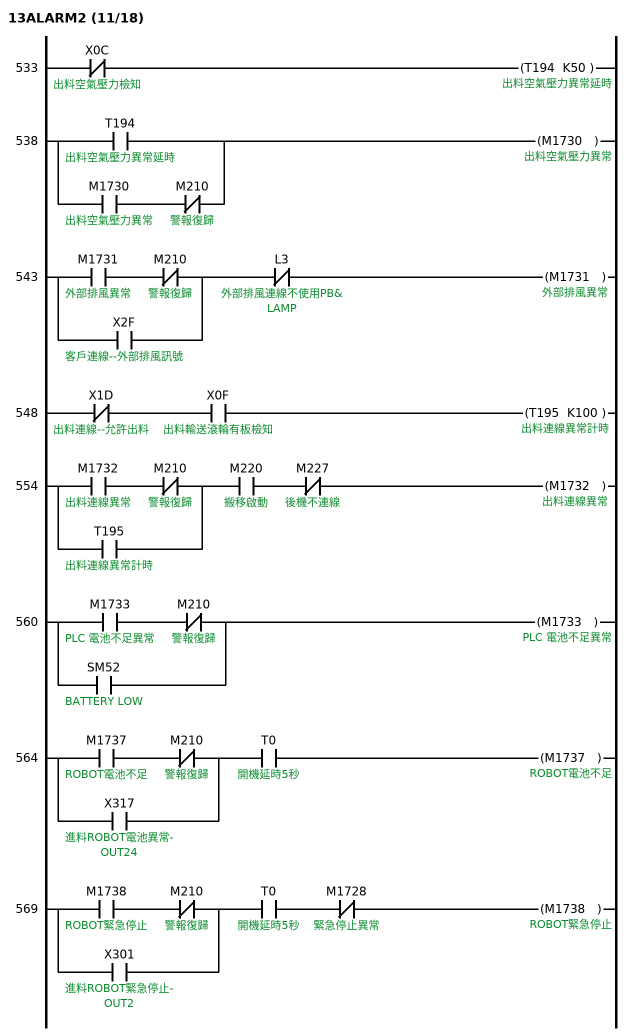
[picture p72: ladder of 13ALARM2, rungs at steps 533 to 569]
533   LDI     X0C  ; 出料空氣壓力檢知
      OUT     T194 K50  ; 出料空氣壓力異常延時
538   LD      T194  ; 出料空氣壓力異常延時
      LD      M1730  ; 出料空氣壓力異常
      ANI     M210  ; 警報復歸
      ORB
      OUT     M1730  ; 出料空氣壓力異常
543   LD      M1731  ; 外部排風異常
      ANI     M210  ; 警報復歸
      OR      X2F  ; 客戶連線--外部排風訊號
      ANI     L3  ; 外部排風連線不使用PB&LAMP
      OUT     M1731  ; 外部排風異常
548   LDI     X1D  ; 出料連線--允許出料
      AND     X0F  ; 出料輸送滾輪有板檢知
      OUT     T195 K100  ; 出料連線異常計時
554   LD      M1732  ; 出料連線異常
      ANI     M210  ; 警報復歸
      OR      T195  ; 出料連線異常計時
      AND     M220  ; 搬移啟動
      ANI     M227  ; 後機不連線
      OUT     M1732  ; 出料連線異常
560   LD      M1733  ; PLC 電池不足異常
      ANI     M210  ; 警報復歸
      OR      SM52  ; BATTERY LOW
      OUT     M1733  ; PLC 電池不足異常
564   LD      M1737  ; ROBOT電池不足
      ANI     M210  ; 警報復歸
      OR      X317  ; 進料ROBOT電池異常-OUT24
      AND     T0  ; 開機延時5秒
      OUT     M1737  ; ROBOT電池不足
569   LD      M1738  ; ROBOT緊急停止
      ANI     M210  ; 警報復歸
      OR      X301  ; 進料ROBOT緊急停止-OUT2
      AND     T0  ; 開機延時5秒
      ANI     M1728  ; 緊急停止異常
      OUT     M1738  ; ROBOT緊急停止
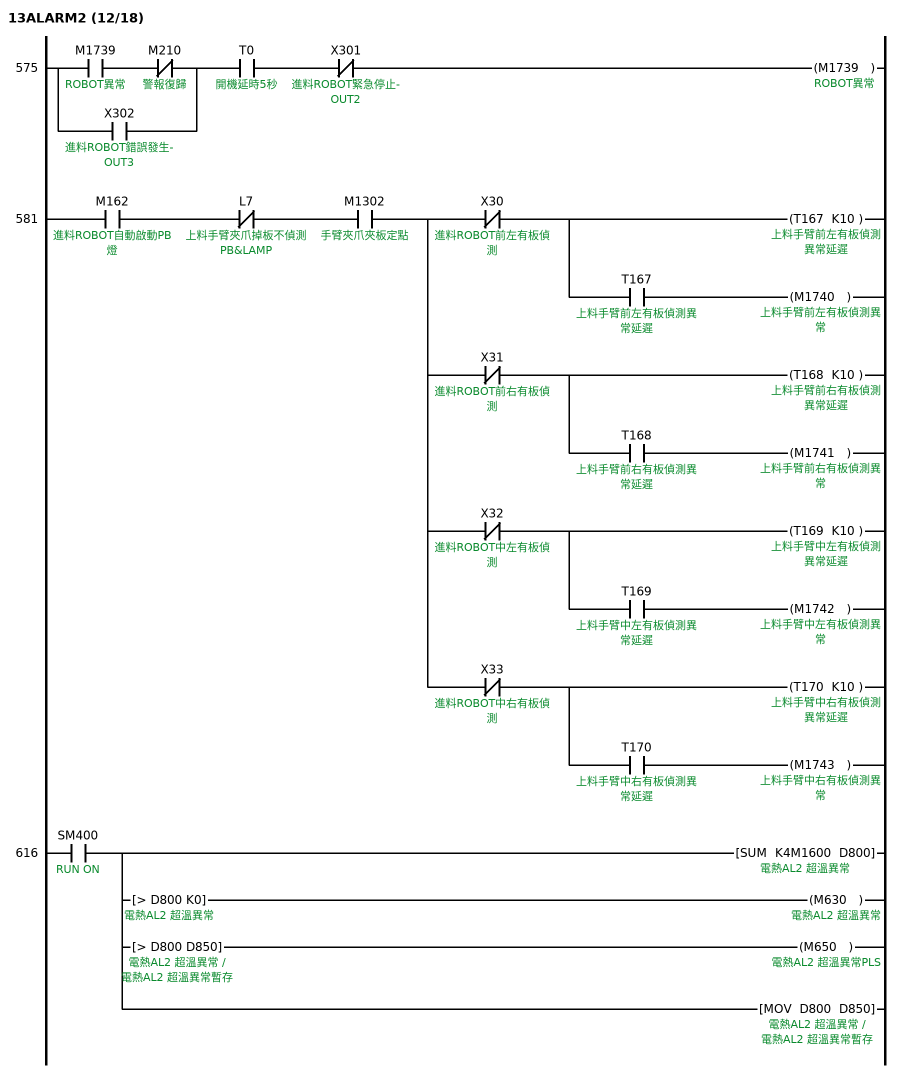
575   LD      M1739  ; ROBOT異常
      ANI     M210  ; 警報復歸
      OR      X302  ; 進料ROBOT錯誤發生-OUT3
      AND     T0  ; 開機延時5秒
      ANI     X301  ; 進料ROBOT緊急停止-OUT2
      OUT     M1739  ; ROBOT異常
581   LD      M162  ; 進料ROBOT自動啟動PB燈
      ANI     L7  ; 上料手臂夾爪掉板不偵測PB&LAMP
      AND     M1302  ; 手臂夾爪夾板定點
      MPS
      ANI     X30  ; 進料ROBOT前左有板偵測
      OUT     T167 K10  ; 上料手臂前左有板偵測異常延遲
      AND     T167  ; 上料手臂前左有板偵測異常延遲
      OUT     M1740  ; 上料手臂前左有板偵測異常
      MRD
      ANI     X31  ; 進料ROBOT前右有板偵測
      OUT     T168 K10  ; 上料手臂前右有板偵測異常延遲
      AND     T168  ; 上料手臂前右有板偵測異常延遲
      OUT     M1741  ; 上料手臂前右有板偵測異常
      MRD
      ANI     X32  ; 進料ROBOT中左有板偵測
      OUT     T169 K10  ; 上料手臂中左有板偵測異常延遲
      AND     T169  ; 上料手臂中左有板偵測異常延遲
      OUT     M1742  ; 上料手臂中左有板偵測異常
      MPP
      ANI     X33  ; 進料ROBOT中右有板偵測
      OUT     T170 K10  ; 上料手臂中右有板偵測異常延遲
      AND     T170  ; 上料手臂中右有板偵測異常延遲
      OUT     M1743  ; 上料手臂中右有板偵測異常
616   LD      SM400  ; RUN ON
      SUM     K4M1600 D800  ; #01 電熱AL2 超溫 / 電熱AL2 超溫異常
      MPS
      AND>    D800 K0  ; 電熱AL2 超溫異常
      OUT     M630  ; 電熱AL2 超溫異常
      MRD
      AND>    D800 D850  ; 電熱AL2 超溫異常 / 電熱AL2 超溫異常暫存
      OUT     M650  ; 電熱AL2 超溫異常PLS
      MPP
      MOV     D800 D850
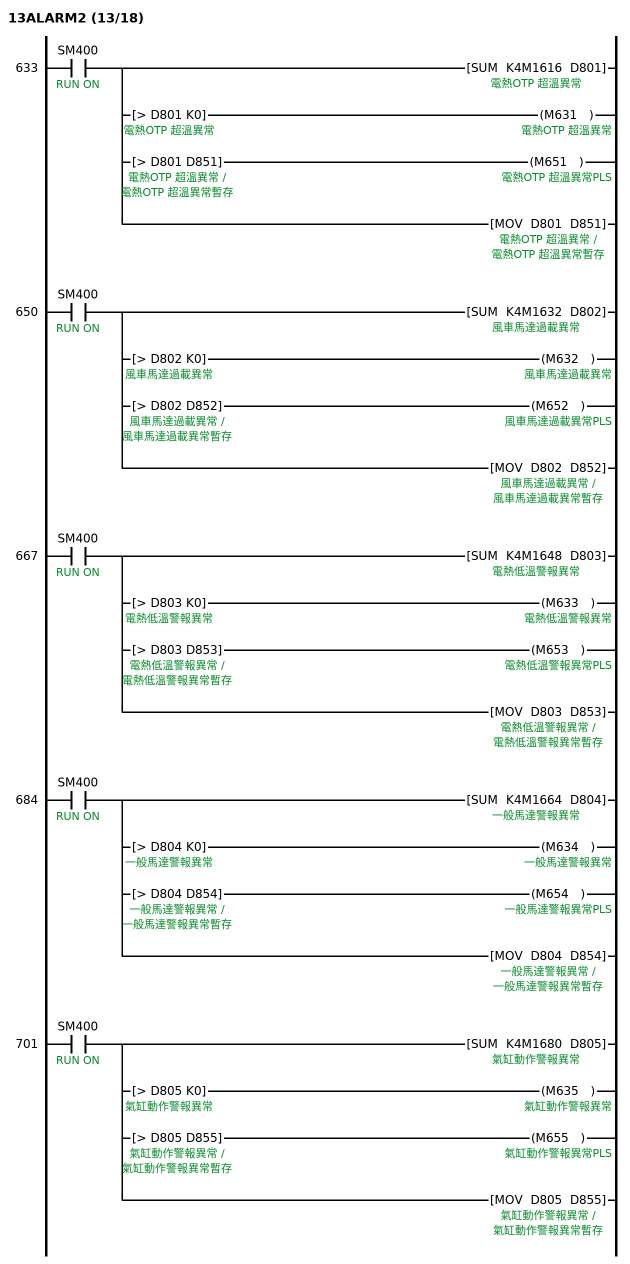
633   LD      SM400  ; RUN ON
      SUM     K4M1616 D801  ; #01 電熱OTP 超溫 / 電熱OTP 超溫異常
      MPS
      AND>    D801 K0  ; 電熱OTP 超溫異常
      OUT     M631  ; 電熱OTP 超溫異常
      MRD
      AND>    D801 D851  ; 電熱OTP 超溫異常 / 電熱OTP 超溫異常暫存
      OUT     M651  ; 電熱OTP 超溫異常PLS
      MPP
      MOV     D801 D851
650   LD      SM400  ; RUN ON
      SUM     K4M1632 D802  ; #01 風車過載 / 風車馬達過載異常
      MPS
      AND>    D802 K0  ; 風車馬達過載異常
      OUT     M632  ; 風車馬達過載異常
      MRD
      AND>    D802 D852  ; 風車馬達過載異常 / 風車馬達過載異常暫存
      OUT     M652  ; 風車馬達過載異常PLS
      MPP
      MOV     D802 D852
667   LD      SM400  ; RUN ON
      SUM     K4M1648 D803  ; #01 低溫警報 / 電熱低溫警報異常
      MPS
      AND>    D803 K0  ; 電熱低溫警報異常
      OUT     M633  ; 電熱低溫警報異常
      MRD
      AND>    D803 D853  ; 電熱低溫警報異常 / 電熱低溫警報異常暫存
      OUT     M653  ; 電熱低溫警報異常PLS
      MPP
      MOV     D803 D853
684   LD      SM400  ; RUN ON
      SUM     K4M1664 D804  ; 一般馬達警報異常
      MPS
      AND>    D804 K0  ; 一般馬達警報異常
      OUT     M634  ; 一般馬達警報異常
      MRD
      AND>    D804 D854  ; 一般馬達警報異常 / 一般馬達警報異常暫存
      OUT     M654  ; 一般馬達警報異常PLS
      MPP
      MOV     D804 D854
701   LD      SM400  ; RUN ON
      SUM     K4M1680 D805  ; 氣缸動作警報異常
      MPS
      AND>    D805 K0  ; 氣缸動作警報異常
      OUT     M635  ; 氣缸動作警報異常
      MRD
      AND>    D805 D855  ; 氣缸動作警報異常 / 氣缸動作警報異常暫存
      OUT     M655  ; 氣缸動作警報異常PLS
      MPP
      MOV     D805 D855
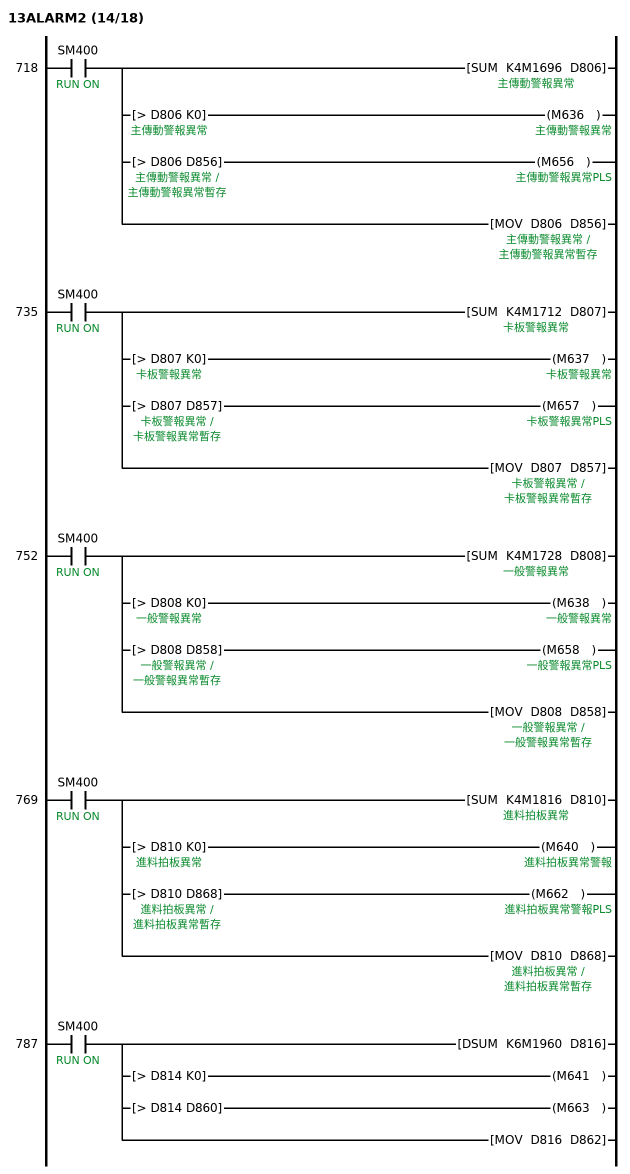
718   LD      SM400  ; RUN ON
      SUM     K4M1696 D806  ; 主傳動警報異常
      MPS
      AND>    D806 K0  ; 主傳動警報異常
      OUT     M636  ; 主傳動警報異常
      MRD
      AND>    D806 D856  ; 主傳動警報異常 / 主傳動警報異常暫存
      OUT     M656  ; 主傳動警報異常PLS
      MPP
      MOV     D806 D856
735   LD      SM400  ; RUN ON
      SUM     K4M1712 D807  ; 卡板警報異常
      MPS
      AND>    D807 K0  ; 卡板警報異常
      OUT     M637  ; 卡板警報異常
      MRD
      AND>    D807 D857  ; 卡板警報異常 / 卡板警報異常暫存
      OUT     M657  ; 卡板警報異常PLS
      MPP
      MOV     D807 D857
752   LD      SM400  ; RUN ON
      SUM     K4M1728 D808  ; 一般警報異常
      MPS
      AND>    D808 K0  ; 一般警報異常
      OUT     M638  ; 一般警報異常
      MRD
      AND>    D808 D858  ; 一般警報異常 / 一般警報異常暫存
      OUT     M658  ; 一般警報異常PLS
      MPP
      MOV     D808 D858
769   LD      SM400  ; RUN ON
      SUM     K4M1816 D810  ; 輸送機輸送變頻器異常-ALM / 進料拍板異常
      MPS
      AND>    D810 K0  ; 進料拍板異常
      OUT     M640  ; 進料拍板異常警報
      MRD
      AND>    D810 D868  ; 進料拍板異常 / 進料拍板異常暫存
      OUT     M662  ; 進料拍板異常警報PLS
      MPP
      MOV     D810 D868
787   LD      SM400  ; RUN ON
      DSUM    K6M1960 D816
      MPS
      AND>    D814 K0
      OUT     M641
      MRD
      AND>    D814 D860
      OUT     M663
      MPP
      MOV     D816 D862
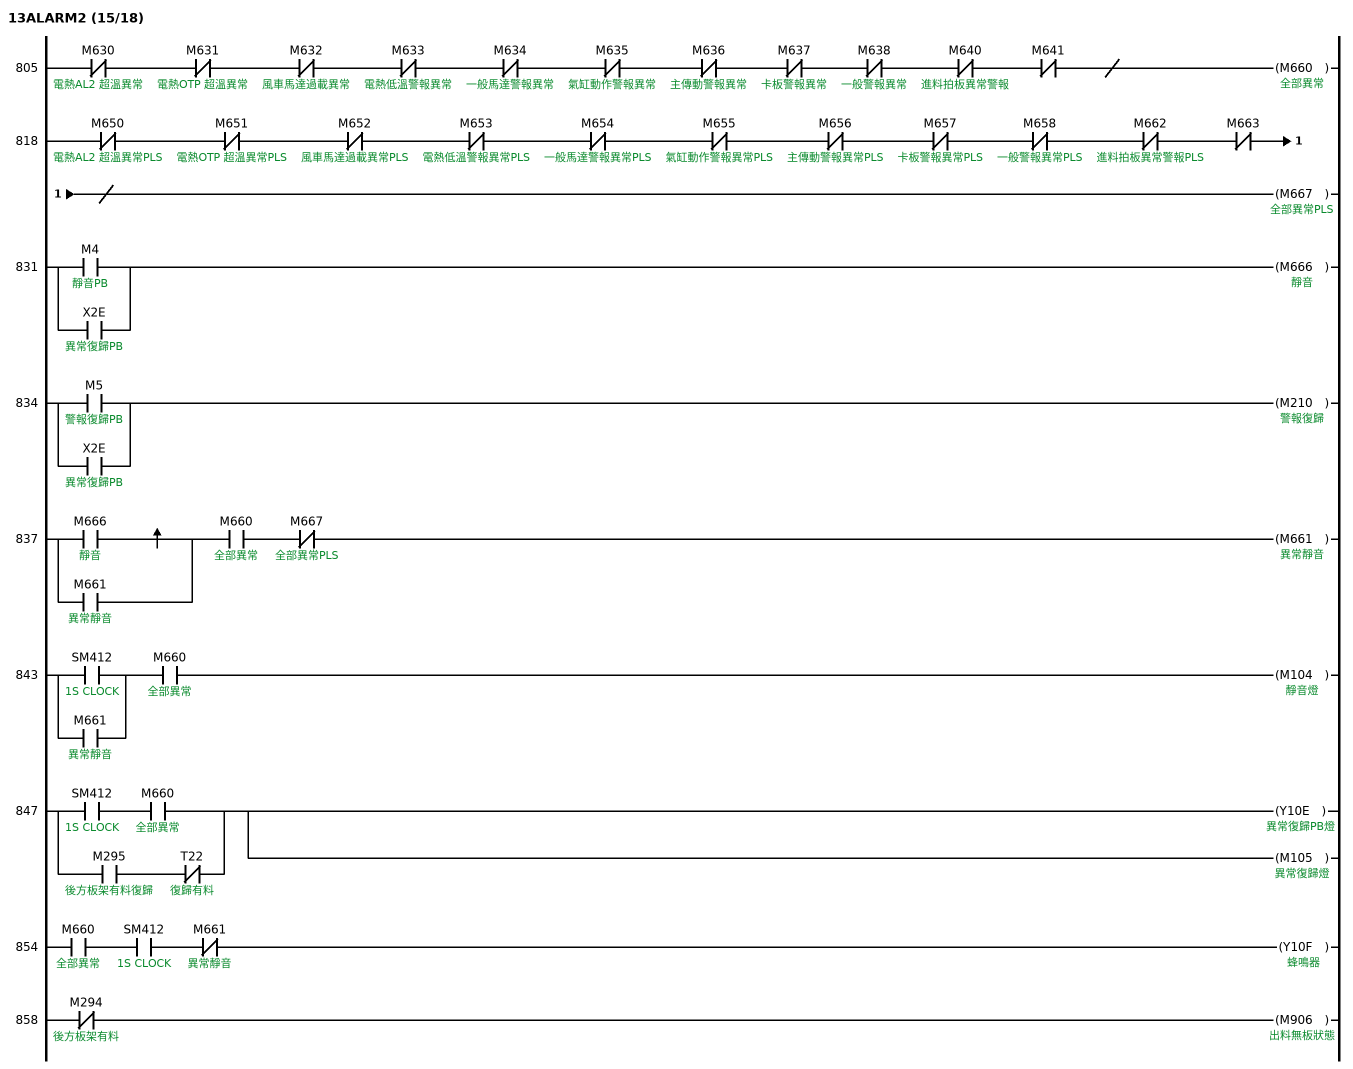
805   LDI     M630  ; 電熱AL2 超溫異常
      ANI     M631  ; 電熱OTP 超溫異常
      ANI     M632  ; 風車馬達過載異常
      ANI     M633  ; 電熱低溫警報異常
      ANI     M634  ; 一般馬達警報異常
      ANI     M635  ; 氣缸動作警報異常
      ANI     M636  ; 主傳動警報異常
      ANI     M637  ; 卡板警報異常
      ANI     M638  ; 一般警報異常
      ANI     M640  ; 進料拍板異常警報
      ANI     M641
      INV
      OUT     M660  ; 全部異常
818   LDI     M650  ; 電熱AL2 超溫異常PLS
      ANI     M651  ; 電熱OTP 超溫異常PLS
      ANI     M652  ; 風車馬達過載異常PLS
      ANI     M653  ; 電熱低溫警報異常PLS
      ANI     M654  ; 一般馬達警報異常PLS
      ANI     M655  ; 氣缸動作警報異常PLS
      ANI     M656  ; 主傳動警報異常PLS
      ANI     M657  ; 卡板警報異常PLS
      ANI     M658  ; 一般警報異常PLS
      ANI     M662  ; 進料拍板異常警報PLS
      ANI     M663
      INV
      OUT     M667  ; 全部異常PLS
831   LD      M4  ; 靜音PB
      OR      X2E  ; 異常復歸PB
      OUT     M666  ; 靜音
834   LD      M5  ; 警報復歸PB
      OR      X2E  ; 異常復歸PB
      OUT     M210  ; 警報復歸
837   LD      M666  ; 靜音
      MEP
      OR      M661  ; 異常靜音
      AND     M660  ; 全部異常
      ANI     M667  ; 全部異常PLS
      OUT     M661  ; 異常靜音
843   LD      SM412  ; 1S CLOCK
      OR      M661  ; 異常靜音
      AND     M660  ; 全部異常
      OUT     M104  ; 靜音燈
847   LD      SM412  ; 1S CLOCK
      AND     M660  ; 全部異常
      LD      M295  ; 後方板架有料復歸
      ANI     T22  ; 復歸有料
      ORB
      OUT     Y10E  ; 異常復歸PB燈
      OUT     M105  ; 異常復歸燈
854   LD      M660  ; 全部異常
      AND     SM412  ; 1S CLOCK
      ANI     M661  ; 異常靜音
      OUT     Y10F  ; 蜂鳴器
858   LDI     M294  ; 後方板架有料
      OUT     M906  ; 出料無板狀態
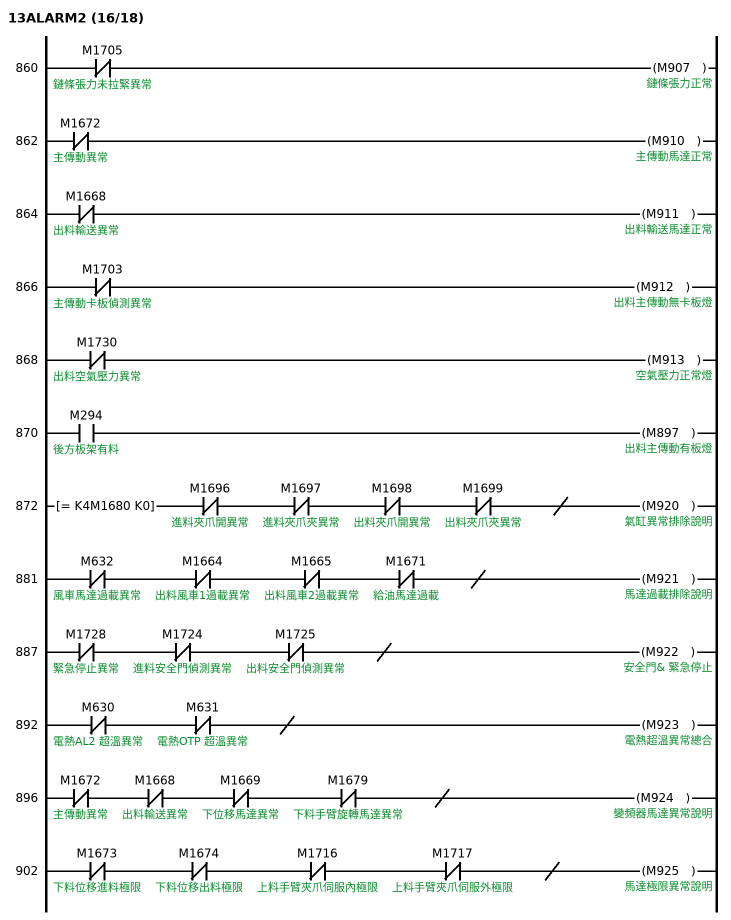
860   LDI     M1705  ; 鏈條張力未拉緊異常
      OUT     M907  ; 鏈條張力正常
862   LDI     M1672  ; 主傳動異常
      OUT     M910  ; 主傳動馬達正常
864   LDI     M1668  ; 出料輸送異常
      OUT     M911  ; 出料輸送馬達正常
866   LDI     M1703  ; 主傳動卡板偵測異常
      OUT     M912  ; 出料主傳動無卡板燈
868   LDI     M1730  ; 出料空氣壓力異常
      OUT     M913  ; 空氣壓力正常燈
870   LD      M294  ; 後方板架有料
      OUT     M897  ; 出料主傳動有板燈
872   LD=     K4M1680 K0  ; 上料手臂前夾爪放異常
      ANI     M1696  ; 進料夾爪開異常
      ANI     M1697  ; 進料夾爪夾異常
      ANI     M1698  ; 出料夾爪開異常
      ANI     M1699  ; 出料夾爪夾異常
      INV
      OUT     M920  ; 氣缸異常排除說明
881   LDI     M632  ; 風車馬達過載異常
      ANI     M1664  ; 出料風車1過載異常
      ANI     M1665  ; 出料風車2過載異常
      ANI     M1671  ; 給油馬達過載
      INV
      OUT     M921  ; 馬達過載排除說明
887   LDI     M1728  ; 緊急停止異常
      ANI     M1724  ; 進料安全門偵測異常
      ANI     M1725  ; 出料安全門偵測異常
      INV
      OUT     M922  ; 安全門& 緊急停止
892   LDI     M630  ; 電熱AL2 超溫異常
      ANI     M631  ; 電熱OTP 超溫異常
      INV
      OUT     M923  ; 電熱超溫異常總合
896   LDI     M1672  ; 主傳動異常
      ANI     M1668  ; 出料輸送異常
      ANI     M1669  ; 下位移馬達異常
      ANI     M1679  ; 下料手臂旋轉馬達異常
      INV
      OUT     M924  ; 變頻器馬達異常說明
902   LDI     M1673  ; 下料位移進料極限
      ANI     M1674  ; 下料位移出料極限
      ANI     M1716  ; 上料手臂夾爪伺服內極限
      ANI     M1717  ; 上料手臂夾爪伺服外極限
      INV
      OUT     M925  ; 馬達極限異常說明
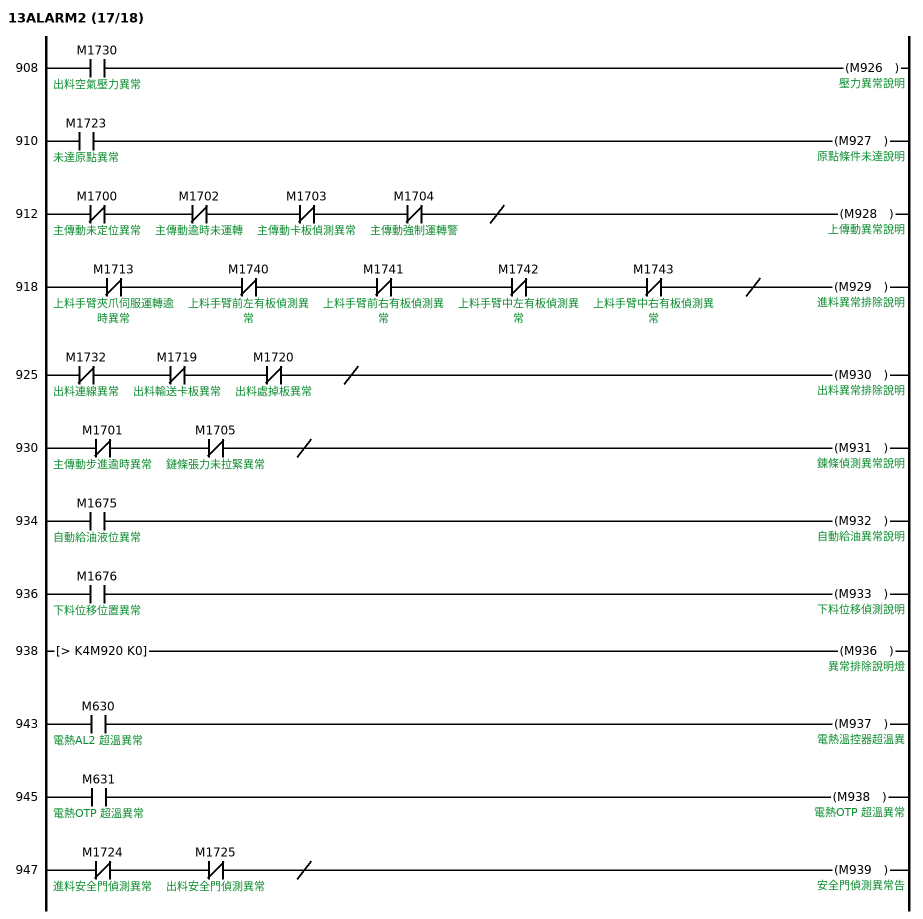
908   LD      M1730  ; 出料空氣壓力異常
      OUT     M926  ; 壓力異常說明
910   LD      M1723  ; 未達原點異常
      OUT     M927  ; 原點條件未達說明
912   LDI     M1700  ; 主傳動未定位異常
      ANI     M1702  ; 主傳動逾時未運轉
      ANI     M1703  ; 主傳動卡板偵測異常
      ANI     M1704  ; 主傳動強制運轉警
      INV
      OUT     M928  ; 上傳動異常說明
918   LDI     M1713  ; 上料手臂夾爪伺服運轉逾時異常
      ANI     M1740  ; 上料手臂前左有板偵測異常
      ANI     M1741  ; 上料手臂前右有板偵測異常
      ANI     M1742  ; 上料手臂中左有板偵測異常
      ANI     M1743  ; 上料手臂中右有板偵測異常
      INV
      OUT     M929  ; 進料異常排除說明
925   LDI     M1732  ; 出料連線異常
      ANI     M1719  ; 出料輸送卡板異常
      ANI     M1720  ; 出料處掉板異常
      INV
      OUT     M930  ; 出料異常排除說明
930   LDI     M1701  ; 主傳動步進逾時異常
      ANI     M1705  ; 鏈條張力未拉緊異常
      INV
      OUT     M931  ; 鍊條偵測異常說明
934   LD      M1675  ; 自動給油液位異常
      OUT     M932  ; 自動給油異常說明
936   LD      M1676  ; 下料位移位置異常
      OUT     M933  ; 下料位移偵測說明
938   LD>     K4M920 K0  ; 氣缸異常排除說明
      OUT     M936  ; 異常排除說明燈
943   LD      M630  ; 電熱AL2 超溫異常
      OUT     M937  ; 電熱溫控器超溫異
945   LD      M631  ; 電熱OTP 超溫異常
      OUT     M938  ; 電熱OTP 超溫異常
947   LDI     M1724  ; 進料安全門偵測異常
      ANI     M1725  ; 出料安全門偵測異常
      INV
      OUT     M939  ; 安全門偵測異常告
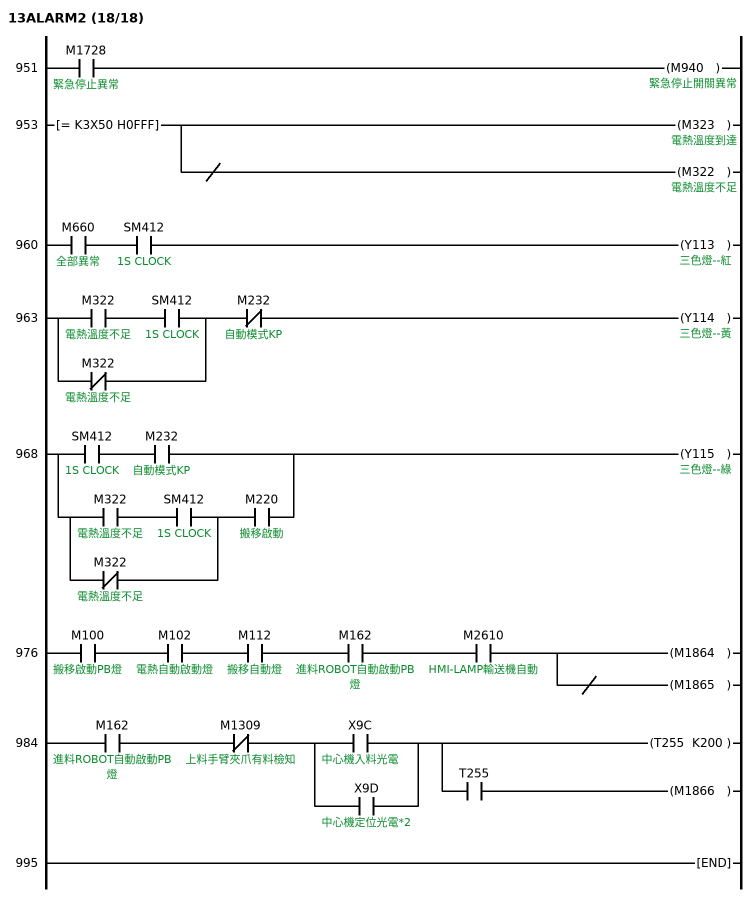
951   LD      M1728  ; 緊急停止異常
      OUT     M940  ; 緊急停止開關異常
953   LD=     K3X50 H0FFF  ; NO,01   溫度到達AL1
      OUT     M323  ; 電熱溫度到達
      INV
      OUT     M322  ; 電熱溫度不足
960   LD      M660  ; 全部異常
      AND     SM412  ; 1S CLOCK
      OUT     Y113  ; 三色燈--紅
963   LD      M322  ; 電熱溫度不足
      AND     SM412  ; 1S CLOCK
      ORI     M322  ; 電熱溫度不足
      ANI     M232  ; 自動模式KP
      OUT     Y114  ; 三色燈--黃
968   LD      SM412  ; 1S CLOCK
      AND     M232  ; 自動模式KP
      LD      M322  ; 電熱溫度不足
      AND     SM412  ; 1S CLOCK
      ORI     M322  ; 電熱溫度不足
      AND     M220  ; 搬移啟動
      ORB
      OUT     Y115  ; 三色燈--綠
976   LD      M100  ; 搬移啟動PB燈
      AND     M102  ; 電熱自動啟動燈
      AND     M112  ; 搬移自動燈
      AND     M162  ; 進料ROBOT自動啟動PB燈
      AND     M2610  ; HMI-LAMP輸送機自動
      OUT     M1864
      INV
      OUT     M1865
984   LD      M162  ; 進料ROBOT自動啟動PB燈
      ANI     M1309  ; 上料手臂夾爪有料檢知
      LD      X9C  ; 中心機入料光電
      OR      X9D  ; 中心機定位光電*2
      ANB
      OUT     T255 K200
      AND     T255
      OUT     M1866
995   END
END_PROGRAM

PROGRAM 14TIME
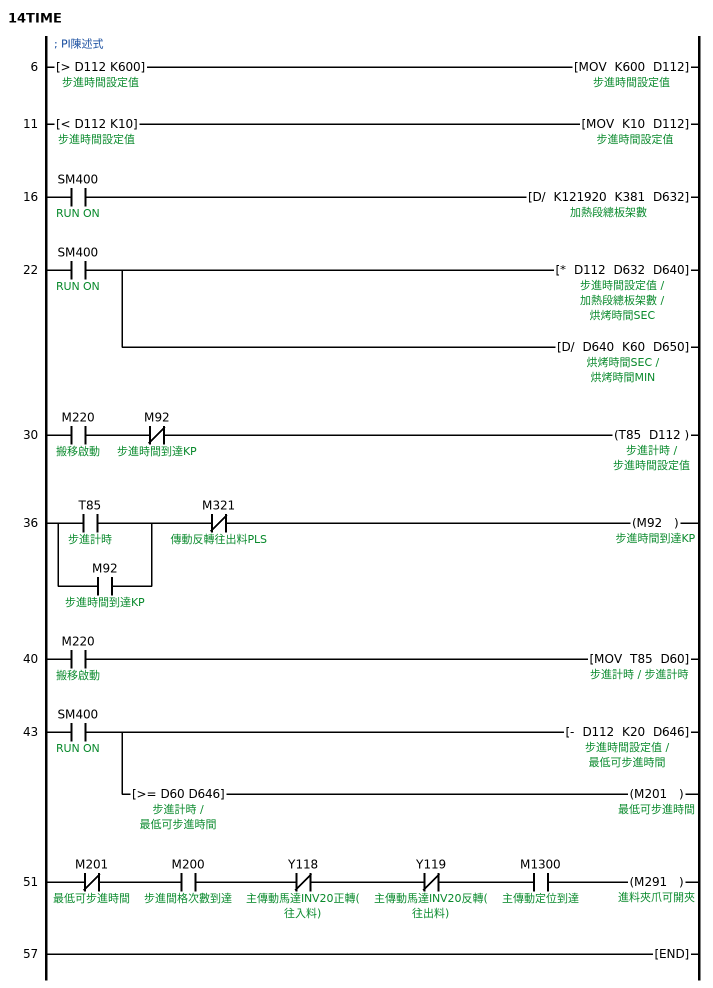
; PI陳述式
6     LD>     D112 K600  ; 步進時間設定值
      MOV     K600 D112
11    LD<     D112 K10  ; 步進時間設定值
      MOV     K10 D112
16    LD      SM400  ; RUN ON
      D/      K121920 K381 D632  ; 加熱段總板架數
22    LD      SM400  ; RUN ON
      *       D112 D632 D640  ; 烘烤時間SEC
      D/      D640 K60 D650  ; 烘烤時間MIN
30    LD      M220  ; 搬移啟動
      ANI     M92  ; 步進時間到達KP
      OUT     T85 D112  ; 步進計時 / 步進時間設定值
36    LD      T85  ; 步進計時
      OR      M92  ; 步進時間到達KP
      ANI     M321  ; 傳動反轉往出料PLS
      OUT     M92  ; 步進時間到達KP
40    LD      M220  ; 搬移啟動
      MOV     T85 D60  ; 步進計時
43    LD      SM400  ; RUN ON
      -       D112 K20 D646  ; 最低可步進時間
      AND>=   D60 D646  ; 步進計時 / 最低可步進時間
      OUT     M201  ; 最低可步進時間
51    LDI     M201  ; 最低可步進時間
      AND     M200  ; 步進間格次數到達
      ANI     Y118  ; 主傳動馬達INV20正轉(往入料)
      ANI     Y119  ; 主傳動馬達INV20反轉(往出料)
      AND     M1300  ; 主傳動定位到達
      OUT     M291  ; 進料夾爪可開夾
57    END
END_PROGRAM

PROGRAM 15STATUS
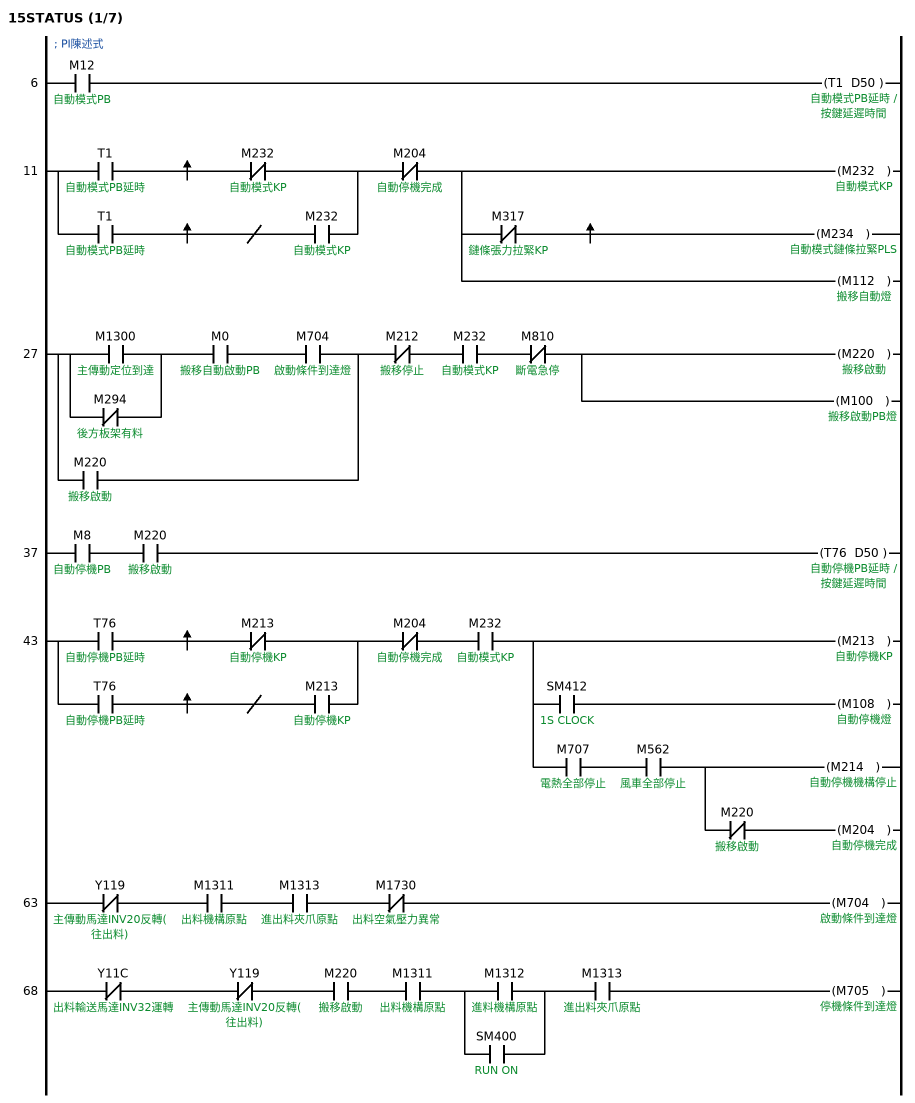
; PI陳述式
6     LD      M12  ; 自動模式PB
      OUT     T1 D50  ; 自動模式PB延時 / 按鍵延遲時間
11    LD      T1  ; 自動模式PB延時
      MEP
      ANI     M232  ; 自動模式KP
      LD      T1  ; 自動模式PB延時
      MEP
      INV
      AND     M232  ; 自動模式KP
      ORB
      ANI     M204  ; 自動停機完成
      OUT     M232  ; 自動模式KP
      MPS
      ANI     M317  ; 鏈條張力拉緊KP
      MEP
      OUT     M234  ; 自動模式鏈條拉緊PLS
      MPP
      OUT     M112  ; 搬移自動燈
27    LD      M1300  ; 主傳動定位到達
      ORI     M294  ; 後方板架有料
      AND     M0  ; 搬移自動啟動PB
      AND     M704  ; 啟動條件到達燈
      OR      M220  ; 搬移啟動
      ANI     M212  ; 搬移停止
      AND     M232  ; 自動模式KP
      ANI     M810  ; 斷電急停
      OUT     M220  ; 搬移啟動
      OUT     M100  ; 搬移啟動PB燈
37    LD      M8  ; 自動停機PB
      AND     M220  ; 搬移啟動
      OUT     T76 D50  ; 自動停機PB延時 / 按鍵延遲時間
43    LD      T76  ; 自動停機PB延時
      MEP
      ANI     M213  ; 自動停機KP
      LD      T76  ; 自動停機PB延時
      MEP
      INV
      AND     M213  ; 自動停機KP
      ORB
      ANI     M204  ; 自動停機完成
      AND     M232  ; 自動模式KP
      OUT     M213  ; 自動停機KP
      MPS
      AND     SM412  ; 1S CLOCK
      OUT     M108  ; 自動停機燈
      MPP
      AND     M707  ; 電熱全部停止
      AND     M562  ; 風車全部停止
      OUT     M214  ; 自動停機機構停止
      ANI     M220  ; 搬移啟動
      OUT     M204  ; 自動停機完成
63    LDI     Y119  ; 主傳動馬達INV20反轉(往出料)
      AND     M1311  ; 出料機構原點
      AND     M1313  ; 進出料夾爪原點
      ANI     M1730  ; 出料空氣壓力異常
      OUT     M704  ; 啟動條件到達燈
68    LDI     Y11C  ; 出料輸送馬達INV32運轉
      ANI     Y119  ; 主傳動馬達INV20反轉(往出料)
      AND     M220  ; 搬移啟動
      AND     M1311  ; 出料機構原點
      LD      M1312  ; 進料機構原點
      OR      SM400  ; RUN ON
      ANB
      AND     M1313  ; 進出料夾爪原點
      OUT     M705  ; 停機條件到達燈
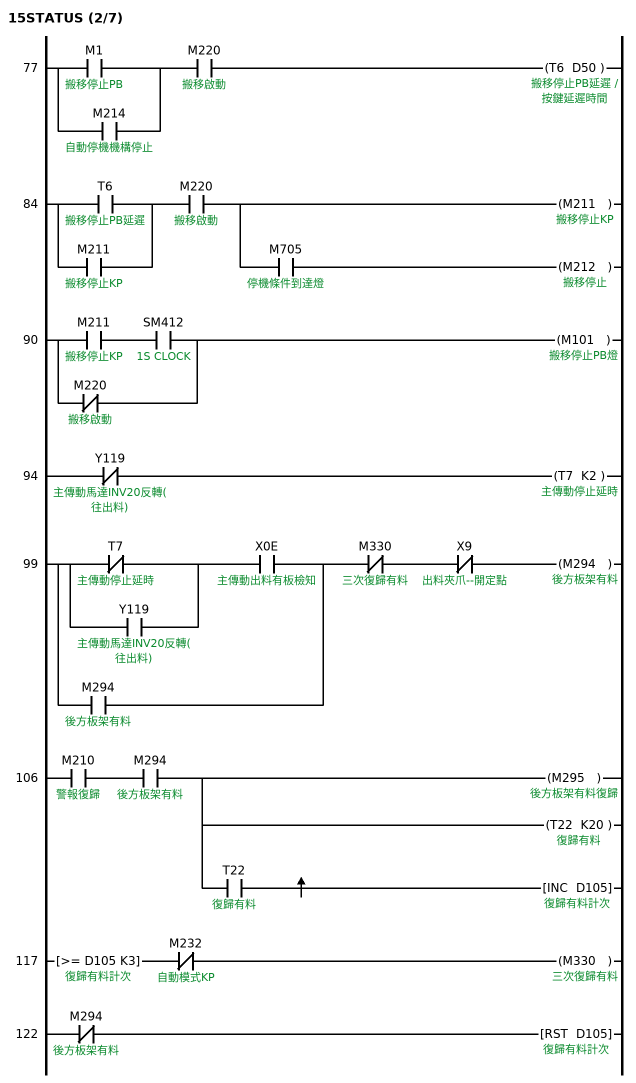
77    LD      M1  ; 搬移停止PB
      OR      M214  ; 自動停機機構停止
      AND     M220  ; 搬移啟動
      OUT     T6 D50  ; 搬移停止PB延遲 / 按鍵延遲時間
84    LD      T6  ; 搬移停止PB延遲
      OR      M211  ; 搬移停止KP
      AND     M220  ; 搬移啟動
      OUT     M211  ; 搬移停止KP
      AND     M705  ; 停機條件到達燈
      OUT     M212  ; 搬移停止
90    LD      M211  ; 搬移停止KP
      AND     SM412  ; 1S CLOCK
      ORI     M220  ; 搬移啟動
      OUT     M101  ; 搬移停止PB燈
94    LDI     Y119  ; 主傳動馬達INV20反轉(往出料)
      OUT     T7 K2  ; 主傳動停止延時
99    LDI     T7  ; 主傳動停止延時
      OR      Y119  ; 主傳動馬達INV20反轉(往出料)
      AND     X0E  ; 主傳動出料有板檢知
      OR      M294  ; 後方板架有料
      ANI     M330  ; 三次復歸有料
      ANI     X9  ; 出料夾爪--開定點
      OUT     M294  ; 後方板架有料
106   LD      M210  ; 警報復歸
      AND     M294  ; 後方板架有料
      OUT     M295  ; 後方板架有料復歸
      OUT     T22 K20  ; 復歸有料
      AND     T22  ; 復歸有料
      MEP
      INC     D105  ; 復歸有料計次
117   LD>=    D105 K3  ; 復歸有料計次
      ANI     M232  ; 自動模式KP
      OUT     M330  ; 三次復歸有料
122   LDI     M294  ; 後方板架有料
      RST     D105  ; 復歸有料計次
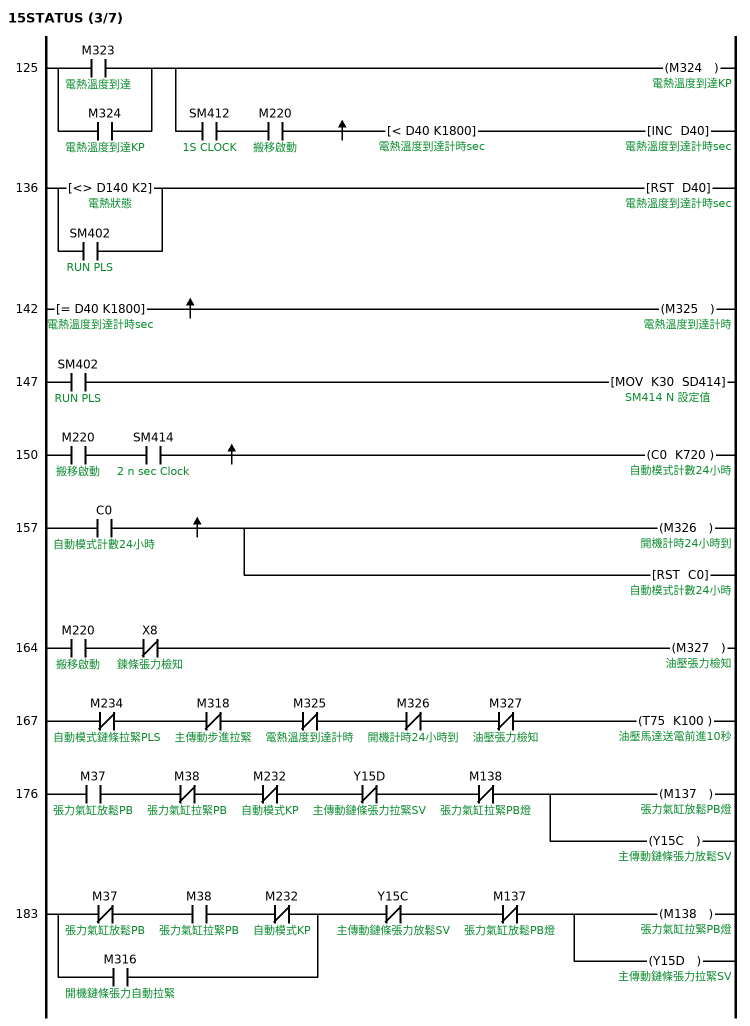
125   LD      M323  ; 電熱溫度到達
      OR      M324  ; 電熱溫度到達KP
      OUT     M324  ; 電熱溫度到達KP
      AND     SM412  ; 1S CLOCK
      AND     M220  ; 搬移啟動
      MEP
      AND<    D40 K1800  ; 電熱溫度到達計時sec
      INC     D40
136   LD<>    D140 K2  ; 電熱狀態
      OR      SM402  ; RUN PLS
      RST     D40  ; 電熱溫度到達計時sec
142   LD=     D40 K1800  ; 電熱溫度到達計時sec
      MEP
      OUT     M325  ; 電熱溫度到達計時
147   LD      SM402  ; RUN PLS
      MOV     K30 SD414  ; SM414 N 設定值
150   LD      M220  ; 搬移啟動
      AND     SM414  ; 2 n sec Clock
      MEP
      OUT     C0 K720  ; 自動模式計數24小時
157   LD      C0  ; 自動模式計數24小時
      MEP
      OUT     M326  ; 開機計時24小時到
      RST     C0  ; 自動模式計數24小時
164   LD      M220  ; 搬移啟動
      ANI     X8  ; 鍊條張力檢知
      OUT     M327  ; 油壓張力檢知
167   LDI     M234  ; 自動模式鏈條拉緊PLS
      ANI     M318  ; 主傳動步進拉緊
      ANI     M325  ; 電熱溫度到達計時
      ANI     M326  ; 開機計時24小時到
      ANI     M327  ; 油壓張力檢知
      OUT     T75 K100  ; 油壓馬達送電前進10秒
176   LD      M37  ; 張力氣缸放鬆PB
      ANI     M38  ; 張力氣缸拉緊PB
      ANI     M232  ; 自動模式KP
      ANI     Y15D  ; 主傳動鏈條張力拉緊SV
      ANI     M138  ; 張力氣缸拉緊PB燈
      OUT     M137  ; 張力氣缸放鬆PB燈
      OUT     Y15C  ; 主傳動鏈條張力放鬆SV
183   LDI     M37  ; 張力氣缸放鬆PB
      AND     M38  ; 張力氣缸拉緊PB
      ANI     M232  ; 自動模式KP
      OR      M316  ; 開機鏈條張力自動拉緊
      ANI     Y15C  ; 主傳動鏈條張力放鬆SV
      ANI     M137  ; 張力氣缸放鬆PB燈
      OUT     M138  ; 張力氣缸拉緊PB燈
      OUT     Y15D  ; 主傳動鏈條張力拉緊SV
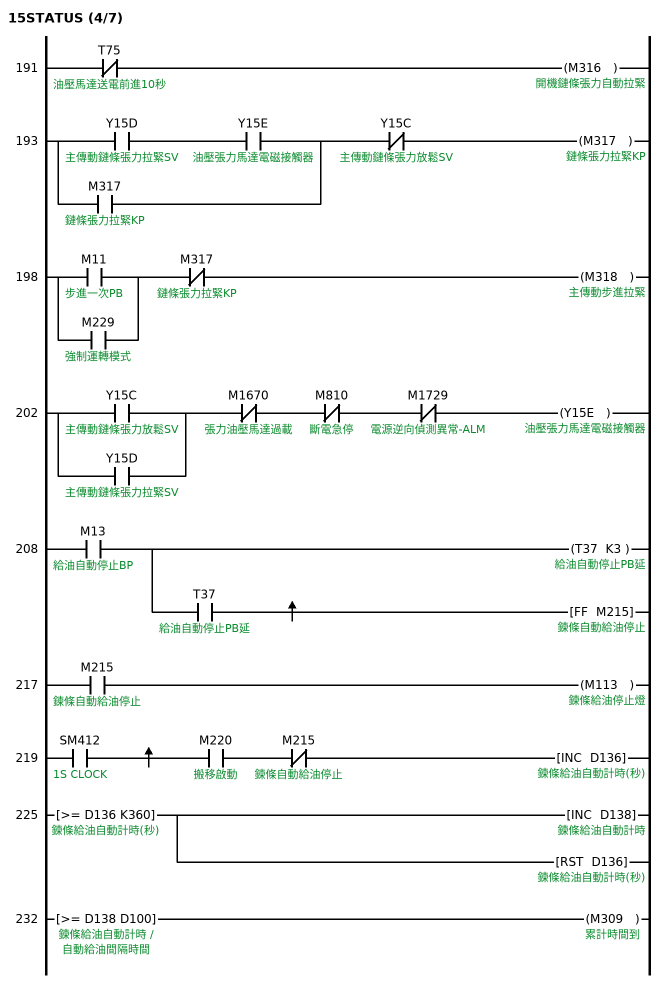
191   LDI     T75  ; 油壓馬達送電前進10秒
      OUT     M316  ; 開機鏈條張力自動拉緊
193   LD      Y15D  ; 主傳動鏈條張力拉緊SV
      AND     Y15E  ; 油壓張力馬達電磁接觸器
      OR      M317  ; 鏈條張力拉緊KP
      ANI     Y15C  ; 主傳動鏈條張力放鬆SV
      OUT     M317  ; 鏈條張力拉緊KP
198   LD      M11  ; 步進一次PB
      OR      M229  ; 強制運轉模式
      ANI     M317  ; 鏈條張力拉緊KP
      OUT     M318  ; 主傳動步進拉緊
202   LD      Y15C  ; 主傳動鏈條張力放鬆SV
      OR      Y15D  ; 主傳動鏈條張力拉緊SV
      ANI     M1670  ; 張力油壓馬達過載
      ANI     M810  ; 斷電急停
      ANI     M1729  ; 電源逆向偵測異常-ALM
      OUT     Y15E  ; 油壓張力馬達電磁接觸器
208   LD      M13  ; 給油自動停止BP
      OUT     T37 K3  ; 給油自動停止PB延
      AND     T37  ; 給油自動停止PB延
      MEP
      FF      M215  ; 鍊條自動給油停止
217   LD      M215  ; 鍊條自動給油停止
      OUT     M113  ; 鍊條給油停止燈
219   LD      SM412  ; 1S CLOCK
      MEP
      AND     M220  ; 搬移啟動
      ANI     M215  ; 鍊條自動給油停止
      INC     D136  ; 鍊條給油自動計時(秒)
225   LD>=    D136 K360  ; 鍊條給油自動計時(秒)
      INC     D138  ; 鍊條給油自動計時
      RST     D136  ; 鍊條給油自動計時(秒)
232   LD>=    D138 D100  ; 鍊條給油自動計時 / 自動給油間隔時間
      OUT     M309  ; 累計時間到
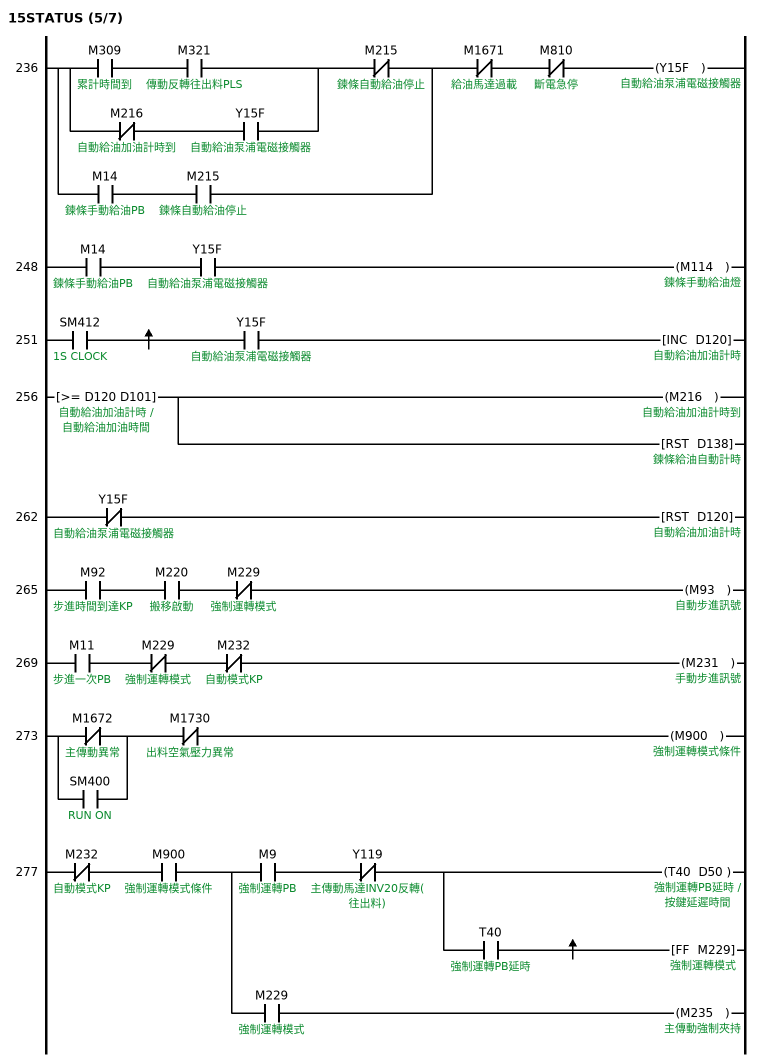
236   LD      M309  ; 累計時間到
      AND     M321  ; 傳動反轉往出料PLS
      LDI     M216  ; 自動給油加油計時到
      AND     Y15F  ; 自動給油泵浦電磁接觸器
      ORB
      ANI     M215  ; 鍊條自動給油停止
      LD      M14  ; 鍊條手動給油PB
      AND     M215  ; 鍊條自動給油停止
      ORB
      ANI     M1671  ; 給油馬達過載
      ANI     M810  ; 斷電急停
      OUT     Y15F  ; 自動給油泵浦電磁接觸器
248   LD      M14  ; 鍊條手動給油PB
      AND     Y15F  ; 自動給油泵浦電磁接觸器
      OUT     M114  ; 鍊條手動給油燈
251   LD      SM412  ; 1S CLOCK
      MEP
      AND     Y15F  ; 自動給油泵浦電磁接觸器
      INC     D120  ; 自動給油加油計時
256   LD>=    D120 D101  ; 自動給油加油計時 / 自動給油加油時間
      OUT     M216  ; 自動給油加油計時到
      RST     D138  ; 鍊條給油自動計時
262   LDI     Y15F  ; 自動給油泵浦電磁接觸器
      RST     D120  ; 自動給油加油計時
265   LD      M92  ; 步進時間到達KP
      AND     M220  ; 搬移啟動
      ANI     M229  ; 強制運轉模式
      OUT     M93  ; 自動步進訊號
269   LD      M11  ; 步進一次PB
      ANI     M229  ; 強制運轉模式
      ANI     M232  ; 自動模式KP
      OUT     M231  ; 手動步進訊號
273   LDI     M1672  ; 主傳動異常
      OR      SM400  ; RUN ON
      ANI     M1730  ; 出料空氣壓力異常
      OUT     M900  ; 強制運轉模式條件
277   LDI     M232  ; 自動模式KP
      AND     M900  ; 強制運轉模式條件
      MPS
      AND     M9  ; 強制運轉PB
      ANI     Y119  ; 主傳動馬達INV20反轉(往出料)
      OUT     T40 D50  ; 強制運轉PB延時 / 按鍵延遲時間
      AND     T40  ; 強制運轉PB延時
      MEP
      FF      M229
      MPP
      AND     M229  ; 強制運轉模式
      OUT     M235  ; 主傳動強制夾持
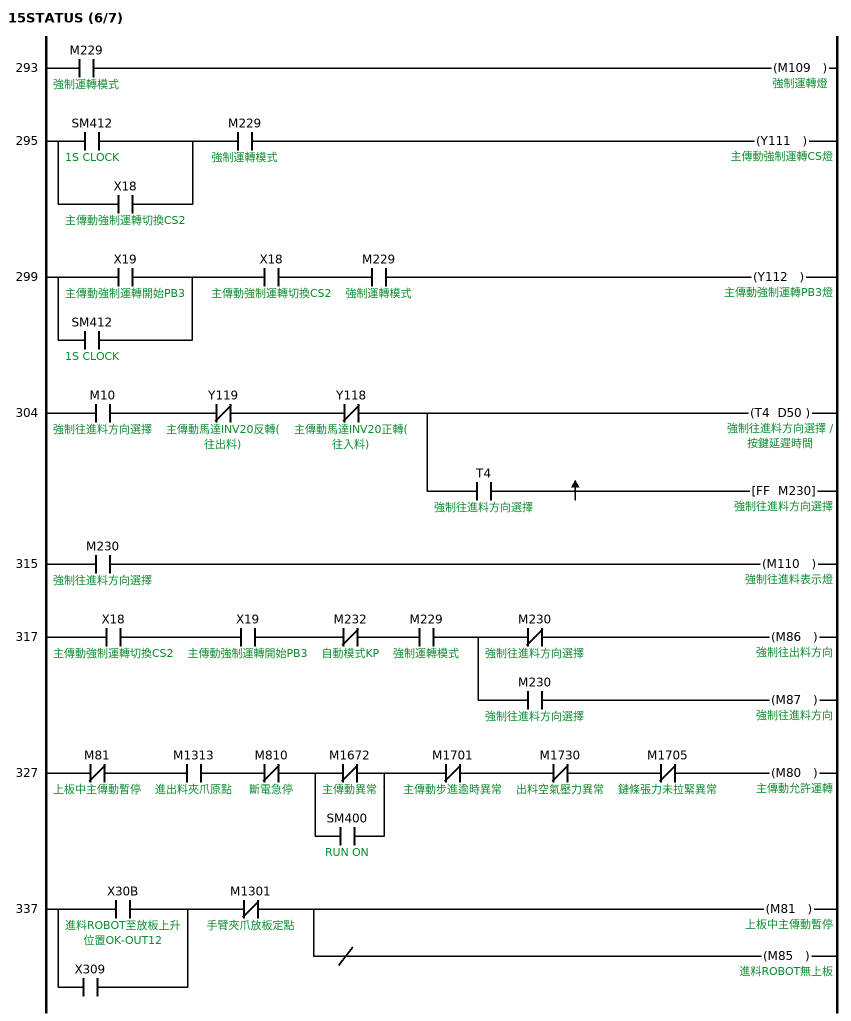
293   LD      M229  ; 強制運轉模式
      OUT     M109  ; 強制運轉燈
295   LD      SM412  ; 1S CLOCK
      OR      X18  ; 主傳動強制運轉切換CS2
      AND     M229  ; 強制運轉模式
      OUT     Y111  ; 主傳動強制運轉CS燈
299   LD      X19  ; 主傳動強制運轉開始PB3
      OR      SM412  ; 1S CLOCK
      AND     X18  ; 主傳動強制運轉切換CS2
      AND     M229  ; 強制運轉模式
      OUT     Y112  ; 主傳動強制運轉PB3燈
304   LD      M10  ; 強制往進料方向選擇
      ANI     Y119  ; 主傳動馬達INV20反轉(往出料)
      ANI     Y118  ; 主傳動馬達INV20正轉(往入料)
      OUT     T4 D50  ; 強制往進料方向選擇 / 按鍵延遲時間
      AND     T4  ; 強制往進料方向選擇
      MEP
      FF      M230  ; 強制往進料方向選擇
315   LD      M230  ; 強制往進料方向選擇
      OUT     M110  ; 強制往進料表示燈
317   LD      X18  ; 主傳動強制運轉切換CS2
      AND     X19  ; 主傳動強制運轉開始PB3
      ANI     M232  ; 自動模式KP
      AND     M229  ; 強制運轉模式
      MPS
      ANI     M230  ; 強制往進料方向選擇
      OUT     M86  ; 強制往出料方向
      MPP
      AND     M230  ; 強制往進料方向選擇
      OUT     M87  ; 強制往進料方向
327   LDI     M81  ; 上板中主傳動暫停
      AND     M1313  ; 進出料夾爪原點
      ANI     M810  ; 斷電急停
      LDI     M1672  ; 主傳動異常
      OR      SM400  ; RUN ON
      ANB
      ANI     M1701  ; 主傳動步進逾時異常
      ANI     M1730  ; 出料空氣壓力異常
      ANI     M1705  ; 鏈條張力未拉緊異常
      OUT     M80  ; 主傳動允許運轉
337   LD      X30B  ; 進料ROBOT至放板上升位置OK-OUT12
      OR      X309
      ANI     M1301  ; 手臂夾爪放板定點
      OUT     M81  ; 上板中主傳動暫停
      INV
      OUT     M85  ; 進料ROBOT無上板
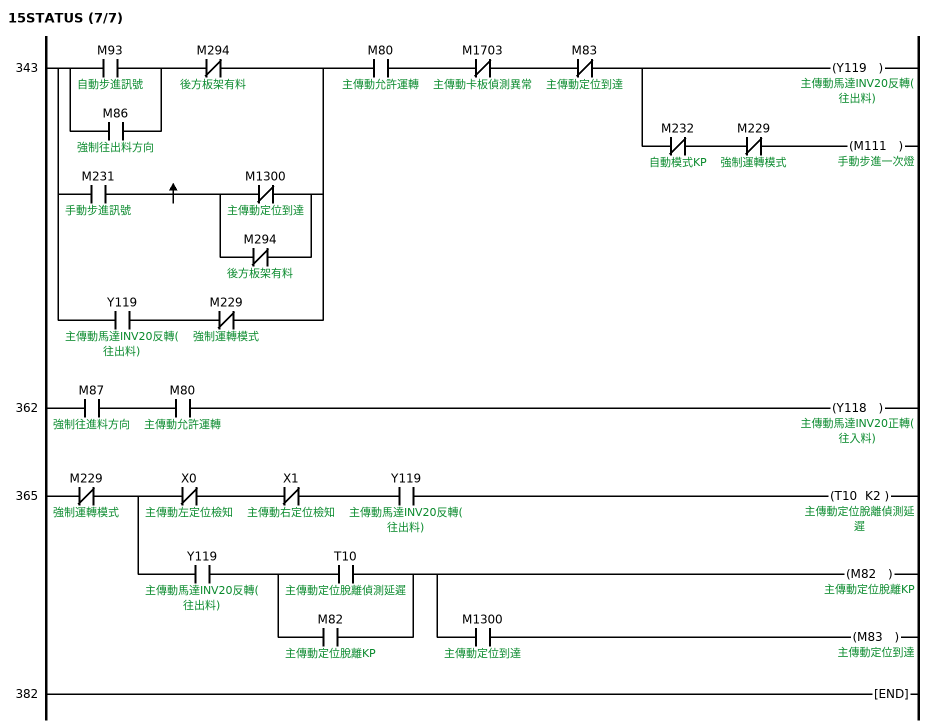
343   LD      M93  ; 自動步進訊號
      OR      M86  ; 強制往出料方向
      ANI     M294  ; 後方板架有料
      LD      M231  ; 手動步進訊號
      MEP
      LDI     M1300  ; 主傳動定位到達
      ORI     M294  ; 後方板架有料
      ANB
      ORB
      LD      Y119  ; 主傳動馬達INV20反轉(往出料)
      ANI     M229  ; 強制運轉模式
      ORB
      AND     M80  ; 主傳動允許運轉
      ANI     M1703  ; 主傳動卡板偵測異常
      ANI     M83  ; 主傳動定位到達
      OUT     Y119  ; 主傳動馬達INV20反轉(往出料)
      ANI     M232  ; 自動模式KP
      ANI     M229  ; 強制運轉模式
      OUT     M111  ; 手動步進一次燈
362   LD      M87  ; 強制往進料方向
      AND     M80  ; 主傳動允許運轉
      OUT     Y118  ; 主傳動馬達INV20正轉(往入料)
365   LDI     M229  ; 強制運轉模式
      MPS
      ANI     X0  ; 主傳動左定位檢知
      ANI     X1  ; 主傳動右定位檢知
      AND     Y119  ; 主傳動馬達INV20反轉(往出料)
      OUT     T10 K2  ; 主傳動定位脫離偵測延遲
      MPP
      AND     Y119  ; 主傳動馬達INV20反轉(往出料)
      LD      T10  ; 主傳動定位脫離偵測延遲
      OR      M82  ; 主傳動定位脫離KP
      ANB
      OUT     M82  ; 主傳動定位脫離KP
      AND     M1300  ; 主傳動定位到達
      OUT     M83  ; 主傳動定位到達
382   END
END_PROGRAM

PROGRAM 16ETHERN
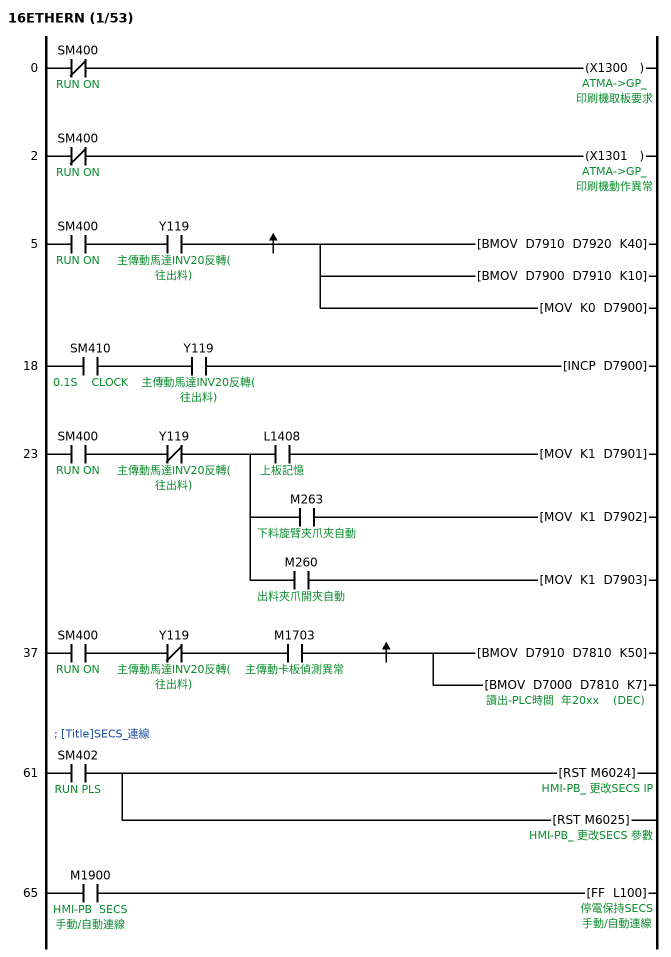
0     LDI     SM400  ; RUN ON
      OUT     X1300  ; ATMA->GP_印刷機取板要求
2     LDI     SM400  ; RUN ON
      OUT     X1301  ; ATMA->GP_印刷機動作異常
5     LD      SM400  ; RUN ON
      AND     Y119  ; 主傳動馬達INV20反轉(往出料)
      MEP
      BMOV    D7910 D7920 K40
      BMOV    D7900 D7910 K10
      MOV     K0 D7900
18    LD      SM410  ; 0.1S    CLOCK
      AND     Y119  ; 主傳動馬達INV20反轉(往出料)
      INCP    D7900
23    LD      SM400  ; RUN ON
      ANI     Y119  ; 主傳動馬達INV20反轉(往出料)
      MPS
      AND     L1408  ; 上板記憶
      MOV     K1 D7901
      MRD
      AND     M263  ; 下料旋臂夾爪夾自動
      MOV     K1 D7902
      MPP
      AND     M260  ; 出料夾爪開夾自動
      MOV     K1 D7903
37    LD      SM400  ; RUN ON
      ANI     Y119  ; 主傳動馬達INV20反轉(往出料)
      AND     M1703  ; 主傳動卡板偵測異常
      MEP
      BMOV    D7910 D7810 K50
      BMOV    D7000 D7810 K7  ; 讀出-PLC時間  年20xx    (DEC)
; [Title]SECS_連線
61    LD      SM402  ; RUN PLS
      RST     M6024  ; HMI-PB_ 更改SECS IP
      RST     M6025  ; HMI-PB_ 更改SECS 參數
65    LD      M1900  ; HMI-PB  SECS    手動/自動連線
      FF      L100  ; 停電保持SECS    手動/自動連線
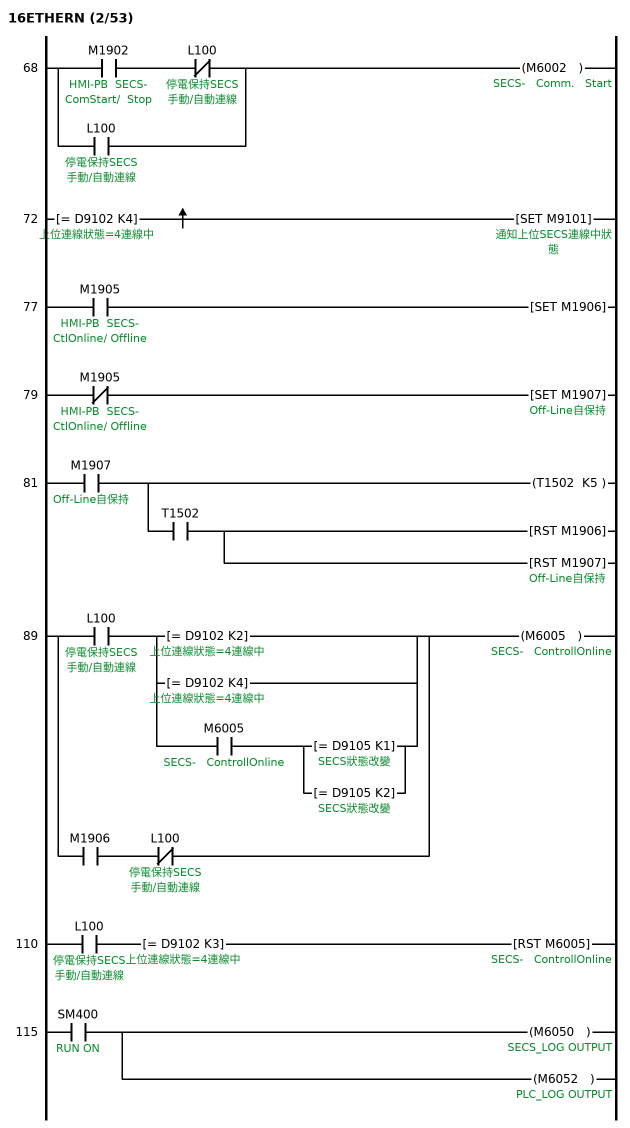
68    LD      M1902  ; HMI-PB  SECS-ComStart/  Stop
      ANI     L100  ; 停電保持SECS    手動/自動連線
      OR      L100  ; 停電保持SECS    手動/自動連線
      OUT     M6002  ; SECS-   Comm.   Start
72    LD=     D9102 K4  ; 上位連線狀態=4連線中
      MEP
      SET     M9101  ; 通知上位SECS連線中狀態
77    LD      M1905  ; HMI-PB  SECS-CtlOnline/ Offline
      SET     M1906
79    LDI     M1905  ; HMI-PB  SECS-CtlOnline/ Offline
      SET     M1907  ; Off-Line自保持
81    LD      M1907  ; Off-Line自保持
      OUT     T1502 K5
      AND     T1502
      RST     M1906
      RST     M1907  ; Off-Line自保持
89    LD      L100  ; 停電保持SECS    手動/自動連線
      LD=     D9102 K2  ; 上位連線狀態=4連線中
      OR=     D9102 K4  ; 上位連線狀態=4連線中
      LD      M6005  ; SECS-   ControllOnline
      LD=     D9105 K1  ; SECS狀態改變
      OR=     D9105 K2  ; SECS狀態改變
      ANB
      ORB
      ANB
      LD      M1906
      ANI     L100  ; 停電保持SECS    手動/自動連線
      ORB
      OUT     M6005  ; SECS-   ControllOnline
110   LD      L100  ; 停電保持SECS    手動/自動連線
      AND=    D9102 K3  ; 上位連線狀態=4連線中
      RST     M6005  ; SECS-   ControllOnline
115   LD      SM400  ; RUN ON
      OUT     M6050  ; SECS_LOG OUTPUT
      OUT     M6052  ; PLC_LOG OUTPUT
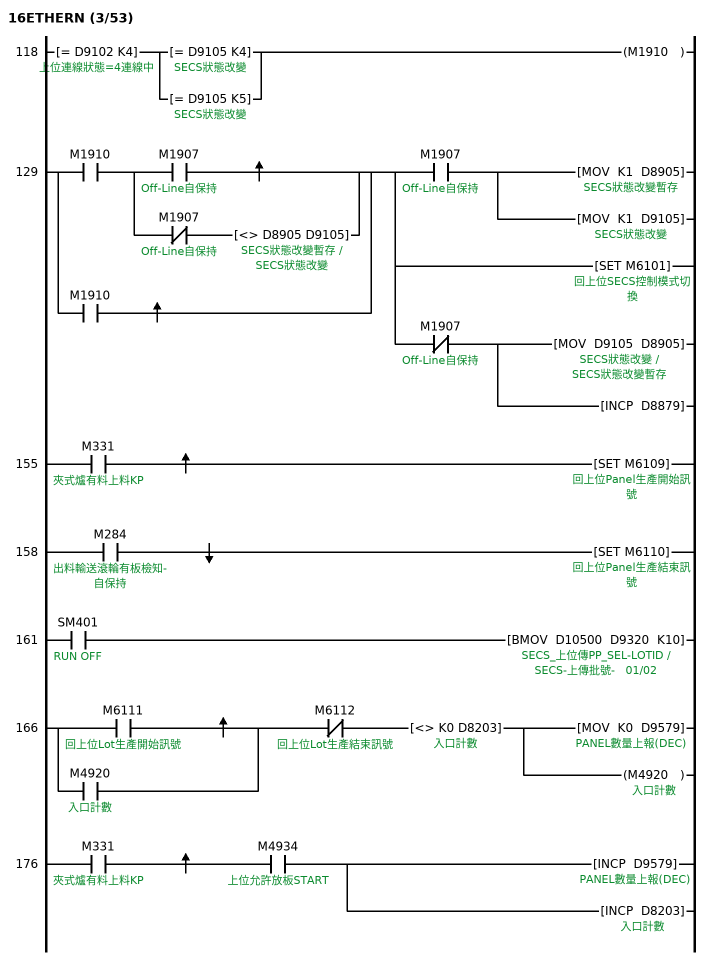
118   LD=     D9102 K4  ; 上位連線狀態=4連線中
      LD=     D9105 K4  ; SECS狀態改變
      OR=     D9105 K5  ; SECS狀態改變
      ANB
      OUT     M1910
129   LD      M1910
      LD      M1907  ; Off-Line自保持
      MEP
      LDI     M1907  ; Off-Line自保持
      AND<>   D8905 D9105  ; SECS狀態改變暫存 / SECS狀態改變
      ORB
      ANB
      LD      M1910
      MEP
      ORB
      MPS
      AND     M1907  ; Off-Line自保持
      MOV     K1 D8905
      MOV     K1 D9105
      MPP
      SET     M6101  ; 回上位SECS控制模式切換
      ANI     M1907  ; Off-Line自保持
      MOV     D9105 D8905
      INCP    D8879
155   LD      M331  ; 夾式爐有料上料KP
      MEP
      SET     M6109  ; 回上位Panel生產開始訊號
158   LD      M284  ; 出料輸送滾輪有板檢知-自保持
      MEF
      SET     M6110  ; 回上位Panel生產結束訊號
161   LD      SM401  ; RUN OFF
      BMOV    D10500 D9320 K10  ; SECS_上位傳PP_SEL-LOTID / SECS-上傳批號-   01/02
166   LD      M6111  ; 回上位Lot生產開始訊號
      MEP
      OR      M4920  ; 入口計數
      ANI     M6112  ; 回上位Lot生產結束訊號
      AND<>   K0 D8203  ; 入口計數
      MOV     K0 D9579  ; PANEL數量上報(DEC)
      OUT     M4920  ; 入口計數
176   LD      M331  ; 夾式爐有料上料KP
      MEP
      AND     M4934  ; 上位允許放板START
      INCP    D9579
      INCP    D8203
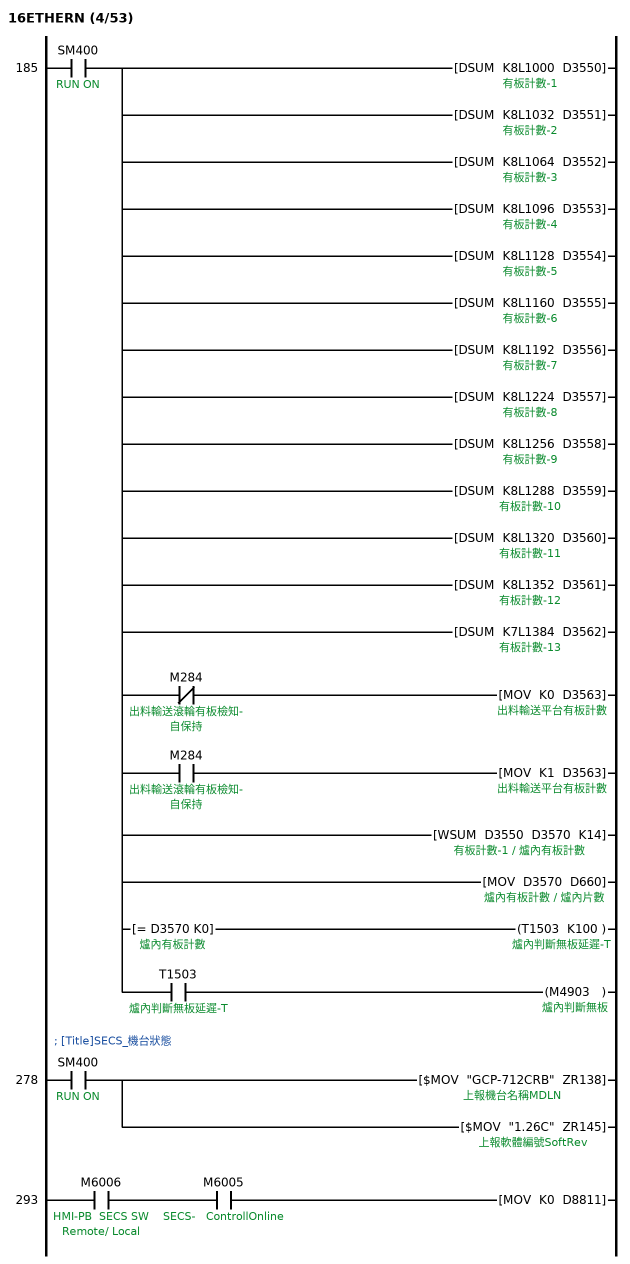
185   LD      SM400  ; RUN ON
      DSUM    K8L1000 D3550  ; 上板記憶 / 有板計數-1
      DSUM    K8L1032 D3551  ; 上板記憶 / 有板計數-2
      DSUM    K8L1064 D3552  ; 上板記憶 / 有板計數-3
      DSUM    K8L1096 D3553  ; 上板記憶 / 有板計數-4
      DSUM    K8L1128 D3554  ; 上板記憶 / 有板計數-5
      DSUM    K8L1160 D3555  ; 上板記憶 / 有板計數-6
      DSUM    K8L1192 D3556  ; 上板記憶 / 有板計數-7
      DSUM    K8L1224 D3557  ; 上板記憶 / 有板計數-8
      DSUM    K8L1256 D3558  ; 上板記憶 / 有板計數-9
      DSUM    K8L1288 D3559  ; 上板記憶 / 有板計數-10
      DSUM    K8L1320 D3560  ; 上板記憶 / 有板計數-11
      DSUM    K8L1352 D3561  ; 上板記憶 / 有板計數-12
      DSUM    K7L1384 D3562  ; 上板記憶 / 有板計數-13
      MPS
      ANI     M284  ; 出料輸送滾輪有板檢知-自保持
      MOV     K0 D3563  ; 出料輸送平台有板計數
      MRD
      AND     M284  ; 出料輸送滾輪有板檢知-自保持
      MOV     K1 D3563
      MPP
      WSUM    D3550 D3570 K14  ; 爐內有板計數
      MOV     D3570 D660  ; 爐內片數
      MPS
      AND=    D3570 K0  ; 爐內有板計數
      OUT     T1503 K100  ; 爐內判斷無板延遲-T
      MPP
      AND     T1503  ; 爐內判斷無板延遲-T
      OUT     M4903  ; 爐內判斷無板
; [Title]SECS_機台狀態
278   LD      SM400  ; RUN ON
      $MOV    "GCP-712CRB" ZR138  ; 上報機台名稱MDLN
      $MOV    "1.26C" ZR145  ; 上報軟體編號SoftRev
293   LD      M6006  ; HMI-PB  SECS SW  Remote/ Local
      AND     M6005  ; SECS-   ControllOnline
      MOV     K0 D8811
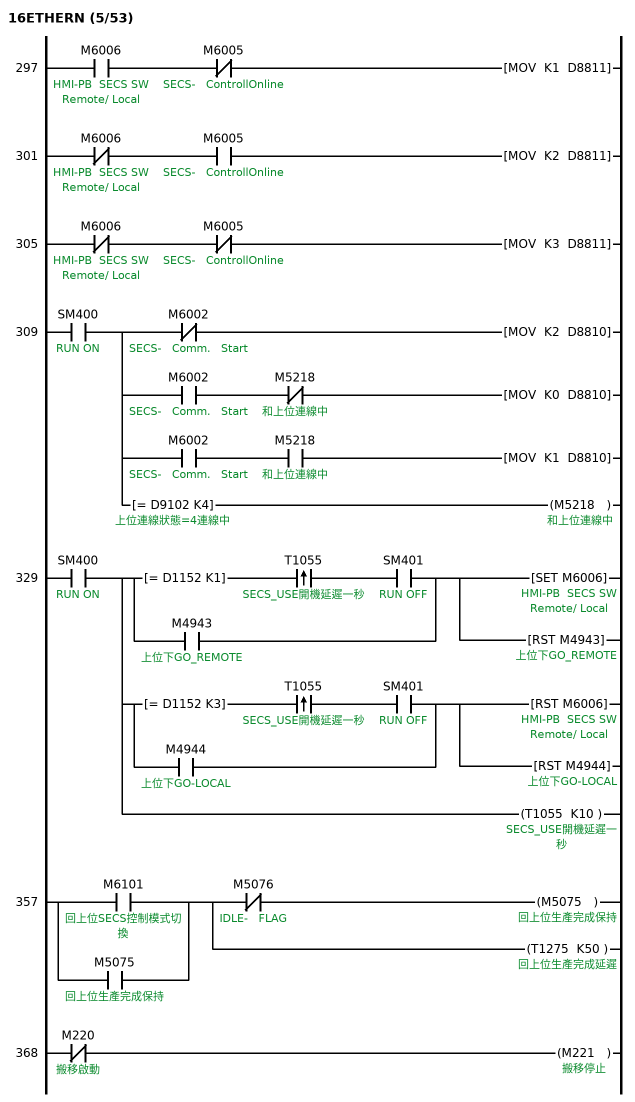
297   LD      M6006  ; HMI-PB  SECS SW  Remote/ Local
      ANI     M6005  ; SECS-   ControllOnline
      MOV     K1 D8811
301   LDI     M6006  ; HMI-PB  SECS SW  Remote/ Local
      AND     M6005  ; SECS-   ControllOnline
      MOV     K2 D8811
305   LDI     M6006  ; HMI-PB  SECS SW  Remote/ Local
      ANI     M6005  ; SECS-   ControllOnline
      MOV     K3 D8811
309   LD      SM400  ; RUN ON
      MPS
      ANI     M6002  ; SECS-   Comm.   Start
      MOV     K2 D8810
      MRD
      AND     M6002  ; SECS-   Comm.   Start
      ANI     M5218  ; 和上位連線中
      MOV     K0 D8810
      MRD
      AND     M6002  ; SECS-   Comm.   Start
      AND     M5218  ; 和上位連線中
      MOV     K1 D8810
      MPP
      AND=    D9102 K4  ; 上位連線狀態=4連線中
      OUT     M5218  ; 和上位連線中
329   LD      SM400  ; RUN ON
      MPS
      LD=     D1152 K1
      ANDP    T1055  ; SECS_USE開機延遲一秒
      AND     SM401  ; RUN OFF
      OR      M4943  ; 上位下GO_REMOTE
      ANB
      SET     M6006  ; HMI-PB  SECS SW  Remote/ Local
      RST     M4943  ; 上位下GO_REMOTE
      MRD
      LD=     D1152 K3
      ANDP    T1055  ; SECS_USE開機延遲一秒
      AND     SM401  ; RUN OFF
      OR      M4944  ; 上位下GO-LOCAL
      ANB
      RST     M6006  ; HMI-PB  SECS SW  Remote/ Local
      RST     M4944  ; 上位下GO-LOCAL
      MPP
      OUT     T1055 K10  ; SECS_USE開機延遲一秒
357   LD      M6101  ; 回上位SECS控制模式切換
      OR      M5075  ; 回上位生產完成保持
      MPS
      ANI     M5076  ; IDLE-   FLAG
      OUT     M5075  ; 回上位生產完成保持
      MPP
      OUT     T1275 K50  ; 回上位生產完成延遲
368   LDI     M220  ; 搬移啟動
      OUT     M221  ; 搬移停止
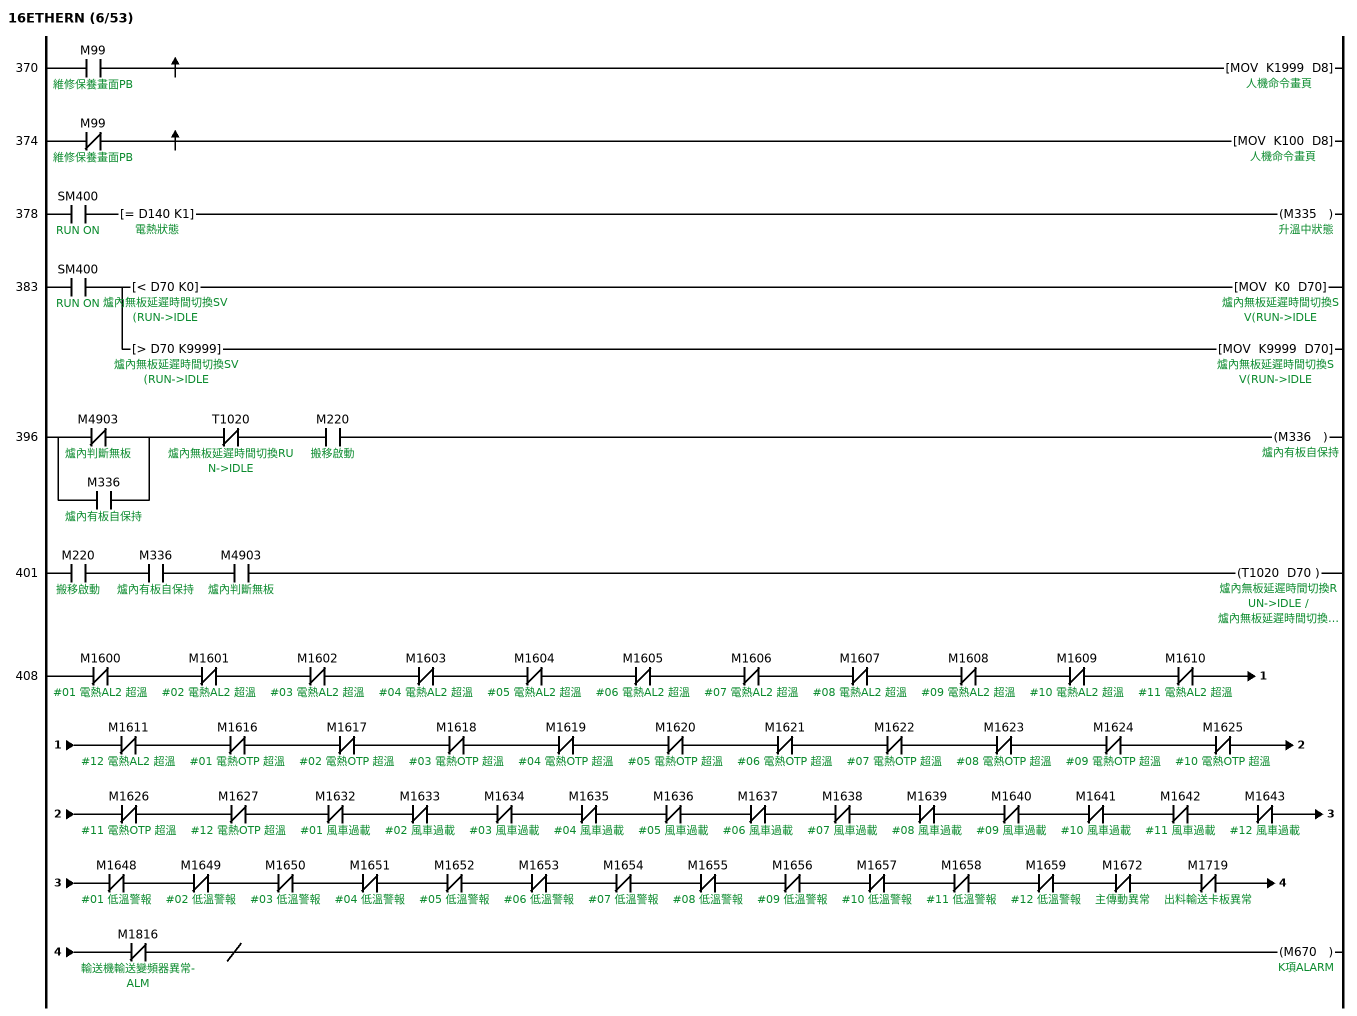
370   LD      M99  ; 維修保養畫面PB
      MEP
      MOV     K1999 D8  ; 人機命令畫頁
374   LDI     M99  ; 維修保養畫面PB
      MEP
      MOV     K100 D8
378   LD      SM400  ; RUN ON
      AND=    D140 K1  ; 電熱狀態
      OUT     M335  ; 升溫中狀態
383   LD      SM400  ; RUN ON
      MPS
      AND<    D70 K0  ; 爐內無板延遲時間切換SV(RUN->IDLE
      MOV     K0 D70
      MPP
      AND>    D70 K9999  ; 爐內無板延遲時間切換SV(RUN->IDLE
      MOV     K9999 D70
396   LDI     M4903  ; 爐內判斷無板
      OR      M336  ; 爐內有板自保持
      ANI     T1020  ; 爐內無板延遲時間切換RUN->IDLE
      AND     M220  ; 搬移啟動
      OUT     M336  ; 爐內有板自保持
401   LD      M220  ; 搬移啟動
      AND     M336  ; 爐內有板自保持
      AND     M4903  ; 爐內判斷無板
      OUT     T1020 D70  ; 爐內無板延遲時間切換RUN->IDLE / 爐內無板延遲時間切換SV(RUN->IDLE
408   LDI     M1600  ; #01 電熱AL2 超溫
      ANI     M1601  ; #02 電熱AL2 超溫
      ANI     M1602  ; #03 電熱AL2 超溫
      ANI     M1603  ; #04 電熱AL2 超溫
      ANI     M1604  ; #05 電熱AL2 超溫
      ANI     M1605  ; #06 電熱AL2 超溫
      ANI     M1606  ; #07 電熱AL2 超溫
      ANI     M1607  ; #08 電熱AL2 超溫
      ANI     M1608  ; #09 電熱AL2 超溫
      ANI     M1609  ; #10 電熱AL2 超溫
      ANI     M1610  ; #11 電熱AL2 超溫
      ANI     M1611  ; #12 電熱AL2 超溫
      ANI     M1616  ; #01 電熱OTP 超溫
      ANI     M1617  ; #02 電熱OTP 超溫
      ANI     M1618  ; #03 電熱OTP 超溫
      ANI     M1619  ; #04 電熱OTP 超溫
      ANI     M1620  ; #05 電熱OTP 超溫
      ANI     M1621  ; #06 電熱OTP 超溫
      ANI     M1622  ; #07 電熱OTP 超溫
      ANI     M1623  ; #08 電熱OTP 超溫
      ANI     M1624  ; #09 電熱OTP 超溫
      ANI     M1625  ; #10 電熱OTP 超溫
      ANI     M1626  ; #11 電熱OTP 超溫
      ANI     M1627  ; #12 電熱OTP 超溫
      ANI     M1632  ; #01 風車過載
      ANI     M1633  ; #02 風車過載
      ANI     M1634  ; #03 風車過載
      ANI     M1635  ; #04 風車過載
      ANI     M1636  ; #05 風車過載
      ANI     M1637  ; #06 風車過載
      ANI     M1638  ; #07 風車過載
      ANI     M1639  ; #08 風車過載
      ANI     M1640  ; #09 風車過載
      ANI     M1641  ; #10 風車過載
      ANI     M1642  ; #11 風車過載
      ANI     M1643  ; #12 風車過載
      ANI     M1648  ; #01 低溫警報
      ANI     M1649  ; #02 低溫警報
      ANI     M1650  ; #03 低溫警報
      ANI     M1651  ; #04 低溫警報
      ANI     M1652  ; #05 低溫警報
      ANI     M1653  ; #06 低溫警報
      ANI     M1654  ; #07 低溫警報
      ANI     M1655  ; #08 低溫警報
      ANI     M1656  ; #09 低溫警報
      ANI     M1657  ; #10 低溫警報
      ANI     M1658  ; #11 低溫警報
      ANI     M1659  ; #12 低溫警報
      ANI     M1672  ; 主傳動異常
      ANI     M1719  ; 出料輸送卡板異常
      ANI     M1816  ; 輸送機輸送變頻器異常-ALM
      INV
      OUT     M670  ; K項ALARM
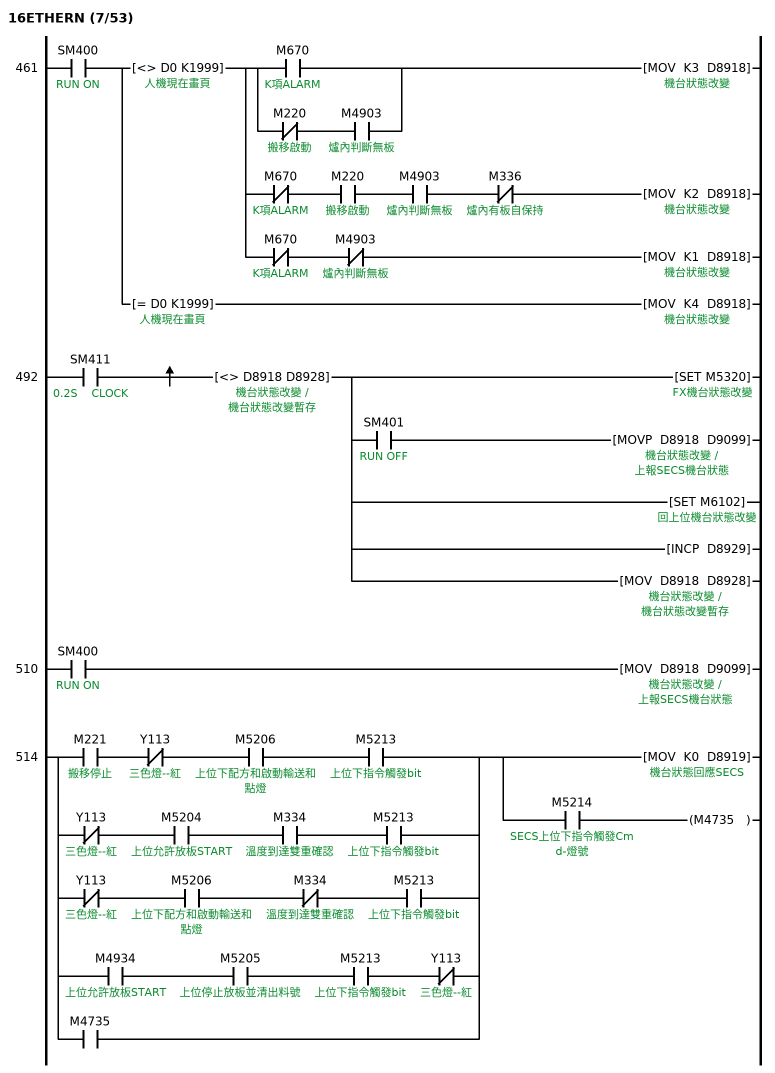
461   LD      SM400  ; RUN ON
      MPS
      AND<>   D0 K1999  ; 人機現在畫頁
      MPS
      LD      M670  ; K項ALARM
      LDI     M220  ; 搬移啟動
      AND     M4903  ; 爐內判斷無板
      ORB
      ANB
      MOV     K3 D8918  ; 機台狀態改變
      MRD
      ANI     M670  ; K項ALARM
      AND     M220  ; 搬移啟動
      AND     M4903  ; 爐內判斷無板
      ANI     M336  ; 爐內有板自保持
      MOV     K2 D8918
      MPP
      ANI     M670  ; K項ALARM
      ANI     M4903  ; 爐內判斷無板
      MOV     K1 D8918
      MPP
      AND=    D0 K1999  ; 人機現在畫頁
      MOV     K4 D8918
492   LD      SM411  ; 0.2S    CLOCK
      MEP
      AND<>   D8918 D8928  ; 機台狀態改變 / 機台狀態改變暫存
      SET     M5320  ; FX機台狀態改變
      MPS
      AND     SM401  ; RUN OFF
      MOVP    D8918 D9099  ; 上報SECS機台狀態
      MPP
      SET     M6102  ; 回上位機台狀態改變
      INCP    D8929
      MOV     D8918 D8928
510   LD      SM400  ; RUN ON
      MOV     D8918 D9099
514   LD      M221  ; 搬移停止
      ANI     Y113  ; 三色燈--紅
      AND     M5206  ; 上位下配方和啟動輸送和點燈
      AND     M5213  ; 上位下指令觸發bit
      LDI     Y113  ; 三色燈--紅
      AND     M5204  ; 上位允許放板START
      AND     M334  ; 溫度到達雙重確認
      AND     M5213  ; 上位下指令觸發bit
      ORB
      LDI     Y113  ; 三色燈--紅
      AND     M5206  ; 上位下配方和啟動輸送和點燈
      ANI     M334  ; 溫度到達雙重確認
      AND     M5213  ; 上位下指令觸發bit
      ORB
      LD      M4934  ; 上位允許放板START
      AND     M5205  ; 上位停止放板並清出料號
      AND     M5213  ; 上位下指令觸發bit
      ANI     Y113  ; 三色燈--紅
      ORB
      OR      M4735
      MOV     K0 D8919  ; 機台狀態回應SECS
      AND     M5214  ; SECS上位下指令觸發Cmd-燈號
      OUT     M4735
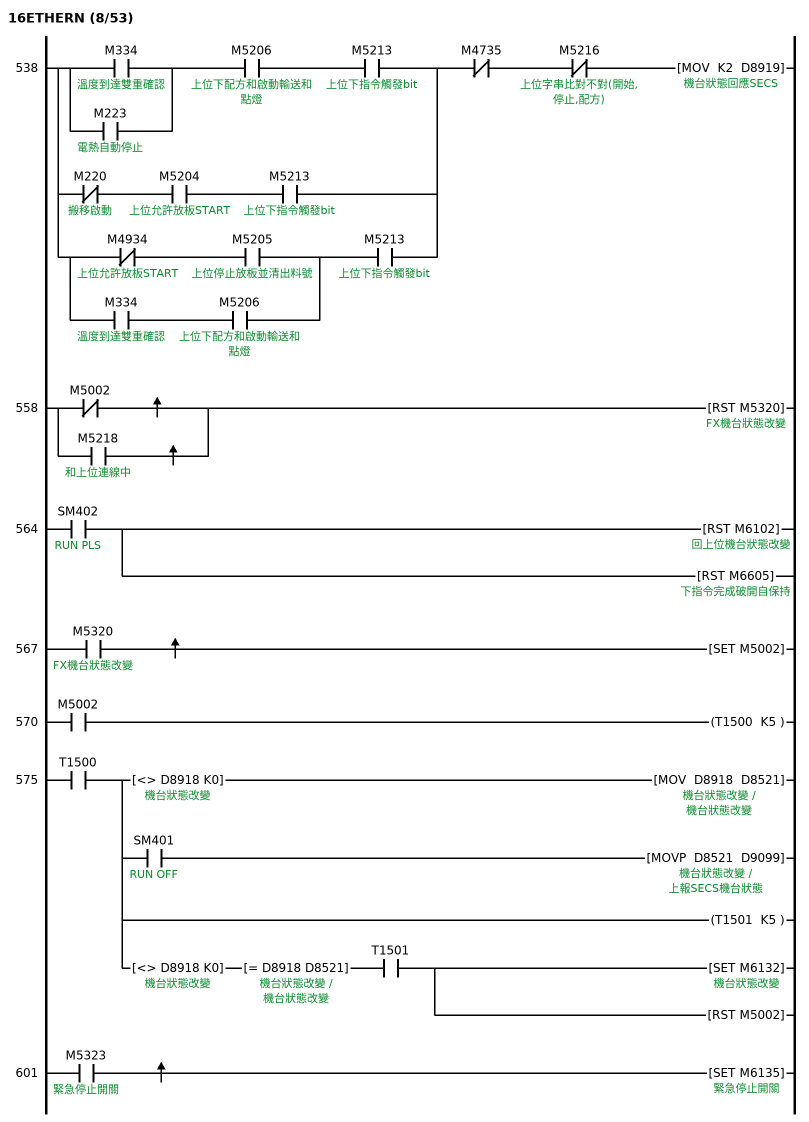
538   LD      M334  ; 溫度到達雙重確認
      OR      M223  ; 電熱自動停止
      AND     M5206  ; 上位下配方和啟動輸送和點燈
      AND     M5213  ; 上位下指令觸發bit
      LDI     M220  ; 搬移啟動
      AND     M5204  ; 上位允許放板START
      AND     M5213  ; 上位下指令觸發bit
      ORB
      LDI     M4934  ; 上位允許放板START
      AND     M5205  ; 上位停止放板並清出料號
      LD      M334  ; 溫度到達雙重確認
      AND     M5206  ; 上位下配方和啟動輸送和點燈
      ORB
      AND     M5213  ; 上位下指令觸發bit
      ORB
      ANI     M4735
      ANI     M5216  ; 上位字串比對不對(開始,停止,配方)
      MOV     K2 D8919
558   LDI     M5002
      MEP
      LD      M5218  ; 和上位連線中
      MEP
      ORB
      RST     M5320  ; FX機台狀態改變
564   LD      SM402  ; RUN PLS
      RST     M6102  ; 回上位機台狀態改變
      RST     M6605  ; 下指令完成破開自保持
567   LD      M5320  ; FX機台狀態改變
      MEP
      SET     M5002
570   LD      M5002
      OUT     T1500 K5
575   LD      T1500
      MPS
      AND<>   D8918 K0  ; 機台狀態改變
      MOV     D8918 D8521  ; 機台狀態改變
      MRD
      AND     SM401  ; RUN OFF
      MOVP    D8521 D9099
      MPP
      OUT     T1501 K5
      AND<>   D8918 K0  ; 機台狀態改變
      AND=    D8918 D8521  ; 機台狀態改變 / 機台狀態改變
      AND     T1501
      SET     M6132  ; 機台狀態改變
      RST     M5002
601   LD      M5323  ; 緊急停止開關
      MEP
      SET     M6135  ; 緊急停止開關
